LIN {X 0,Y 131.837,Z 270.712,A -85,B 0,C 180,E1 -26196.961,E2 -26196.961} C_VEL
LIN {X 0,Y 133.527,Z 251.929,A -85,B 0,C 180,E1 -26198.085,E2 -26198.085} C_VEL
LIN {X 0,Y 135.598,Z 225.127,A -85,B 0,C 180,E1 -26199.486,E2 -26199.486} C_VEL
LIN {X 0,Y 130.645,Z 212.931,A -85,B 0,C 180,E1 -26202.013,E2 -26202.013} C_VEL
LIN {X 0,Y 122.665,Z 198.092,A -85,B 0,C 180,E1 -26206.231,E2 -26206.231} C_VEL
LIN {X 0,Y 115.926,Z 187.635,A -85,B 0,C 180,E1 -26210.225,E2 -26210.225} C_VEL
LIN {X 0,Y 113.416,Z 183.95,A -85,B 0,C 180,E1 -26211.866,E2 -26211.866} C_VEL
LIN {X 0,Y 111.206,Z 180.453,A -85,B 0,C 180,E1 -26213.445,E2 -26213.445} C_VEL
LIN {X 0,Y 108.659,Z 177.597,A -85,B 0,C 180,E1 -26215.273,E2 -26215.273} C_VEL
LIN {X 0,Y 107.799,Z 175.056,A -85,B 0,C 180,E1 -26216.159,E2 -26216.159} C_VEL
LIN {X 0,Y 107.779,Z 175.058,A -85,B 0,C 180,E1 -26222.039,E2 -26222.039} C_VEL
LIN {X 0,Y 107.684,Z 175.066,A -85,B 0,C 180,E1 -26228.449,E2 -26228.449} C_VEL
LIN {X 0,Y 107.678,Z 175.072,A -85,B 0,C 180,E1 -26235.886,E2 -26235.886} C_VEL
LIN {X 0,Y 107.705,Z 175.047,A -85,B 0,C 180,E1 -26241.538,E2 -26241.538} C_VEL
LIN {X 0,Y 107.802,Z 175.038,A -85,B 0,C 180,E1 -26248.565,E2 -26248.565} C_VEL
LIN {X 0,Y 107.911,Z 175.043,A -85,B 0,C 180,E1 -26256.999,E2 -26256.999} C_VEL
LIN {X 0,Y 108.039,Z 175.012,A -85,B 0,C 180,E1 -26264.919,E2 -26264.919} C_VEL
LIN {X 0,Y 108.288,Z 174.994,A -85,B 0,C 180,E1 -26268.773,E2 -26268.773} C_VEL
LIN {X 0,Y 108.457,Z 174.961,A -85,B 0,C 180,E1 -26276.285,E2 -26276.285} C_VEL
LIN {X 0,Y 108.945,Z 174.908,A -85,B 0,C 180,E1 -26280.001,E2 -26280.001} C_VEL
LIN {X 0,Y 108.329,Z 174.987,A -85,B 0,C 180,E1 -26287.456,E2 -26287.456} C_VEL
LIN {X 0,Y 108.2,Z 174.989,A -85,B 0,C 180,E1 -26293.017,E2 -26293.017} C_VEL
LIN {X 0,Y 107.908,Z 175.033,A -85,B 0,C 180,E1 -26299.006,E2 -26299.006} C_VEL
LIN {X 0,Y 107.848,Z 175.044,A -85,B 0,C 180,E1 -26305.296,E2 -26305.296} C_VEL
LIN {X 0,Y 107.812,Z 175.158,A -85,B 0,C 180,E1 -26305.994,E2 -26305.994} C_VEL
LIN {X 0,Y 108.749,Z 177.876,A -85,B 0,C 180,E1 -26306.897,E2 -26306.897} C_VEL
LIN {X 0,Y 110.862,Z 180.069,A -85,B 0,C 180,E1 -26308.39,E2 -26308.39} C_VEL
LIN {X 0,Y 113.377,Z 183.974,A -85,B 0,C 180,E1 -26310.189,E2 -26310.189} C_VEL
LIN {X 0,Y 116.979,Z 189.548,A -85,B 0,C 180,E1 -26312.553,E2 -26312.553} C_VEL
LIN {X 0,Y 121.423,Z 196.893,A -85,B 0,C 180,E1 -26315.224,E2 -26315.224} C_VEL
LIN {X 0,Y 126.867,Z 209.823,A -85,B 0,C 180,E1 -26318.489,E2 -26318.489} C_VEL
LIN {X 0,Y 131.896,Z 223.796,A -85,B 0,C 180,E1 -26321.338,E2 -26321.338} C_VEL
LIN {X 0,Y 133.622,Z 229.369,A -85,B 0,C 180,E1 -26322.318,E2 -26322.318} C_VEL
LIN {X 0,Y 134.484,Z 244.81,A -85,B 0,C 180,E1 -26323.749,E2 -26323.749} C_VEL
LIN {X 0,Y 131.522,Z 280.67,A -85,B 0,C 180,E1 -26325.705,E2 -26325.705} C_VEL
LIN {X 0,Y 129.707,Z 293.105,A -85,B 0,C 180,E1 -26326.838,E2 -26326.838} C_VEL
LIN {X 0,Y 126.95,Z 306.45,A -85,B 0,C 180,E1 -26328.634,E2 -26328.634} C_VEL
LIN {X 0,Y 123.797,Z 318.083,A -85,B 0,C 180,E1 -26330.834,E2 -26330.834} C_VEL
LIN {X 0,Y 120.243,Z 329.412,A -85,B 0,C 180,E1 -26333.716,E2 -26333.716} C_VEL
LIN {X 0,Y 116.614,Z 339.667,A -85,B 0,C 180,E1 -26337.153,E2 -26337.153} C_VEL
LIN {X 0,Y 113.178,Z 348.906,A -85,B 0,C 180,E1 -26341.233,E2 -26341.233} C_VEL
LIN {X 0,Y 109.944,Z 357.92,A -85,B 0,C 180,E1 -26346.452,E2 -26346.452} C_VEL
LIN {X 0,Y 107.523,Z 365.11,A -85,B 0,C 180,E1 -26351.912,E2 -26351.912} C_VEL
LIN {X 0,Y 105.953,Z 371.622,A -85,B 0,C 180,E1 -26358.522,E2 -26358.522} C_VEL
LIN {X 0,Y 105.611,Z 375.867,A -85,B 0,C 180,E1 -26364.271,E2 -26364.271} C_VEL
LIN {X 0,Y 105.837,Z 378.956,A -85,B 0,C 180,E1 -26370,E2 -26370} C_VEL
LIN {X 0,Y 105.526,Z 380.371,A -85,B 0,C 180,E1 -26373.818,E2 -26373.818} C_VEL
LIN {X 0,Y 105.444,Z 381.376,A -85,B 0,C 180,E1 -26377.66,E2 -26377.66} C_VEL
LIN {X 0,Y 106.579,Z 382.189,A -85,B 0,C 180,E1 -26385.293,E2 -26385.293} C_VEL
LIN {X 0,Y 109.574,Z 381.541,A -85,B 0,C 180,E1 -26392.633,E2 -26392.633} C_VEL
LIN {X 0,Y 114.392,Z 379.409,A -85,B 0,C 180,E1 -26399.439,E2 -26399.439} C_VEL
LIN {X 0,Y 120.75,Z 375.708,A -85,B 0,C 180,E1 -26405.593,E2 -26405.593} C_VEL
LIN {X 0,Y 126.372,Z 371.837,A -85,B 0,C 180,E1 -26409.758,E2 -26409.758} C_VEL
LIN {X 0,Y 132.761,Z 366.913,A -85,B 0,C 180,E1 -26413.486,E2 -26413.486} C_VEL
LIN {X 0,Y 140.925,Z 359.728,A -85,B 0,C 180,E1 -26417.357,E2 -26417.357} C_VEL
LIN {X 0,Y 148.839,Z 351.65,A -85,B 0,C 180,E1 -26420.348,E2 -26420.348} C_VEL
LIN {X 0,Y 156.514,Z 342.43,A -85,B 0,C 180,E1 -26422.847,E2 -26422.847} C_VEL
LIN {X 0,Y 163.463,Z 332.667,A -85,B 0,C 180,E1 -26424.774,E2 -26424.774} C_VEL
LIN {X 0,Y 165.572,Z 329.353,A -85,B 0,C 180,E1 -26425.287,E2 -26425.287} C_VEL
LIN {X 0,Y 168.177,Z 324.681,A -85,B 0,C 180,E1 -26426.147,E2 -26426.147} C_VEL
LIN {X 0,Y 171.358,Z 317.027,A -85,B 0,C 180,E1 -26427.987,E2 -26427.987} C_VEL
LIN {X 0,Y 174.237,Z 309.028,A -85,B 0,C 180,E1 -26429.66,E2 -26429.66} C_VEL
LIN {X 0,Y 176.217,Z 303.822,A -85,B 0,C 180,E1 -26430.28,E2 -26430.28} C_VEL
LIN {X 0,Y 180.185,Z 292.508,A -85,B 0,C 180,E1 -26431,E2 -26431} C_VEL
LIN {X 0,Y 183.545,Z 279.289,A -85,B 0,C 180,E1 -26431.581,E2 -26431.581} C_VEL
LIN {X 0,Y 184.874,Z 271.488,A -85,B 0,C 180,E1 -26431.877,E2 -26431.877} C_VEL
LIN {X 0,Y 184.085,Z 267.5,A -85,B 0,C 180,E1 -26434.147,E2 -26434.147} C_VEL
LIN {X 0,Y 183.505,Z 264.746,A -85,B 0,C 180,E1 -26436.214,E2 -26436.214} C_VEL
LIN {X 0,Y 183.071,Z 262.291,A -85,B 0,C 180,E1 -26438.789,E2 -26438.789} C_VEL
LIN {X 0,Y 182.897,Z 261.223,A -85,B 0,C 180,E1 -26441.141,E2 -26441.141} C_VEL
LIN {X 0,Y 183.287,Z 261.303,A -85,B 0,C 180,E1 -26445.419,E2 -26445.419} C_VEL
LIN {X 0,Y 184.804,Z 265.34,A -85,B 0,C 180,E1 -26450.463,E2 -26450.463} C_VEL
LIN {X 0,Y 185.328,Z 267.395,A -85,B 0,C 180,E1 -26451.844,E2 -26451.844} C_VEL
LIN {X 0,Y 182.72,Z 280.977,A -85,B 0,C 180,E1 -26452.43,E2 -26452.43} C_VEL
LIN {X 0,Y 179.105,Z 293.413,A -85,B 0,C 180,E1 -26453.239,E2 -26453.239} C_VEL
LIN {X 0,Y 174.048,Z 306.258,A -85,B 0,C 180,E1 -26454.437,E2 -26454.437} C_VEL
LIN {X 0,Y 168.223,Z 317.797,A -85,B 0,C 180,E1 -26455.895,E2 -26455.895} C_VEL
LIN {X 0,Y 161.224,Z 328.841,A -85,B 0,C 180,E1 -26457.736,E2 -26457.736} C_VEL
LIN {X 0,Y 154.617,Z 337.56,A -85,B 0,C 180,E1 -26459.691,E2 -26459.691} C_VEL
LIN {X 0,Y 146.318,Z 346.778,A -85,B 0,C 180,E1 -26462.502,E2 -26462.502} C_VEL
LIN {X 0,Y 137.818,Z 354.628,A -85,B 0,C 180,E1 -26465.853,E2 -26465.853} C_VEL
LIN {X 0,Y 130.525,Z 360.305,A -85,B 0,C 180,E1 -26469.295,E2 -26469.295} C_VEL
LIN {X 0,Y 122.931,Z 365.24,A -85,B 0,C 180,E1 -26473.619,E2 -26473.619} C_VEL
LIN {X 0,Y 117.561,Z 368.123,A -85,B 0,C 180,E1 -26477.391,E2 -26477.391} C_VEL
LIN {X 0,Y 112.094,Z 370.491,A -85,B 0,C 180,E1 -26482.097,E2 -26482.097} C_VEL
LIN {X 0,Y 107.426,Z 371.92,A -85,B 0,C 180,E1 -26487.254,E2 -26487.254} C_VEL
LIN {X 0,Y 102.613,Z 372.423,A -85,B 0,C 180,E1 -26494.727,E2 -26494.727} C_VEL
LIN {X 0,Y 100.442,Z 371.896,A -85,B 0,C 180,E1 -26499.676,E2 -26499.676} C_VEL
LIN {X 0,Y 98.797,Z 370.594,A -85,B 0,C 180,E1 -26505.344,E2 -26505.344} C_VEL
LIN {X 0,Y 97.987,Z 368.076,A -85,B 0,C 180,E1 -26512.088,E2 -26512.088} C_VEL
LIN {X 0,Y 98.357,Z 364.286,A -85,B 0,C 180,E1 -26519.029,E2 -26519.029} C_VEL
LIN {X 0,Y 99.859,Z 358.869,A -85,B 0,C 180,E1 -26526.194,E2 -26526.194} C_VEL
LIN {X 0,Y 102.179,Z 351.971,A -85,B 0,C 180,E1 -26532.88,E2 -26532.88} C_VEL
LIN {X 0,Y 105.096,Z 344.444,A -85,B 0,C 180,E1 -26538.427,E2 -26538.427} C_VEL
LIN {X 0,Y 108.652,Z 335.44,A -85,B 0,C 180,E1 -26543.501,E2 -26543.501} C_VEL
LIN {X 0,Y 111.955,Z 326.806,A -85,B 0,C 180,E1 -26547.252,E2 -26547.252} C_VEL
LIN {X 0,Y 115.723,Z 316.032,A -85,B 0,C 180,E1 -26550.87,E2 -26550.87} C_VEL
LIN {X 0,Y 119.401,Z 303.884,A -85,B 0,C 180,E1 -26553.946,E2 -26553.946} C_VEL
LIN {X 0,Y 122.429,Z 291.632,A -85,B 0,C 180,E1 -26556.21,E2 -26556.21} C_VEL
LIN {X 0,Y 124.862,Z 278.393,A -85,B 0,C 180,E1 -26557.988,E2 -26557.988} C_VEL
LIN {X 0,Y 126.521,Z 265.545,A -85,B 0,C 180,E1 -26559.089,E2 -26559.089} C_VEL
LIN {X 0,Y 129.685,Z 227.021,A -85,B 0,C 180,E1 -26561.204,E2 -26561.204} C_VEL
LIN {X 0,Y 125.719,Z 217.007,A -85,B 0,C 180,E1 -26563.389,E2 -26563.389} C_VEL
LIN {X 0,Y 118.24,Z 202.715,A -85,B 0,C 180,E1 -26567.693,E2 -26567.693} C_VEL
LIN {X 0,Y 111.077,Z 191.405,A -85,B 0,C 180,E1 -26572.311,E2 -26572.311} C_VEL
LIN {X 0,Y 107.022,Z 185.413,A -85,B 0,C 180,E1 -26575.35,E2 -26575.35} C_VEL
LIN {X 0,Y 104.709,Z 182.294,A -85,B 0,C 180,E1 -26577.202,E2 -26577.202} C_VEL
LIN {X 0,Y 104.052,Z 181.117,A -85,B 0,C 180,E1 -26577.789,E2 -26577.789} C_VEL
LIN {X 0,Y 101.854,Z 179.084,A -85,B 0,C 180,E1 -26579.609,E2 -26579.609} C_VEL
LIN {X 0,Y 100.819,Z 176.566,A -85,B 0,C 180,E1 -26580.74,E2 -26580.74} C_VEL
LIN {X 0,Y 100.71,Z 175.936,A -85,B 0,C 180,E1 -26580.977,E2 -26580.977} C_VEL
LIN {X 0,Y 100.662,Z 175.944,A -85,B 0,C 180,E1 -26583.955,E2 -26583.955} C_VEL
LIN {X 0,Y 100.635,Z 175.933,A -85,B 0,C 180,E1 -26589.809,E2 -26589.809} C_VEL
LIN {X 0,Y 100.648,Z 175.947,A -85,B 0,C 180,E1 -26595.712,E2 -26595.712} C_VEL
LIN {X 0,Y 100.642,Z 175.924,A -85,B 0,C 180,E1 -26601.063,E2 -26601.063} C_VEL
LIN {X 0,Y 100.697,Z 175.936,A -85,B 0,C 180,E1 -26606.879,E2 -26606.879} C_VEL
LIN {X 0,Y 100.786,Z 175.928,A -85,B 0,C 180,E1 -26615.268,E2 -26615.268} C_VEL
LIN {X 0,Y 100.818,Z 175.909,A -85,B 0,C 180,E1 -26619.602,E2 -26619.602} C_VEL
LIN {X 0,Y 101.188,Z 175.879,A -85,B 0,C 180,E1 -26627.974,E2 -26627.974} C_VEL
LIN {X 0,Y 101.267,Z 175.844,A -85,B 0,C 180,E1 -26632.022,E2 -26632.022} C_VEL
LIN {X 0,Y 101.869,Z 175.788,A -85,B 0,C 180,E1 -26640.001,E2 -26640.001} C_VEL
LIN {X 0,Y 101.267,Z 175.868,A -85,B 0,C 180,E1 -26647.979,E2 -26647.979} C_VEL
LIN {X 0,Y 101.125,Z 175.87,A -85,B 0,C 180,E1 -26653.353,E2 -26653.353} C_VEL
LIN {X 0,Y 100.848,Z 176.055,A -85,B 0,C 180,E1 -26661.328,E2 -26661.328} C_VEL
LIN {X 0,Y 101.616,Z 178.356,A -85,B 0,C 180,E1 -26662.225,E2 -26662.225} C_VEL
LIN {X 0,Y 103.667,Z 180.769,A -85,B 0,C 180,E1 -26664.003,E2 -26664.003} C_VEL
LIN {X 0,Y 104.515,Z 181.953,A -85,B 0,C 180,E1 -26664.72,E2 -26664.72} C_VEL
LIN {X 0,Y 106.599,Z 185.091,A -85,B 0,C 180,E1 -26666.426,E2 -26666.426} C_VEL
LIN {X 0,Y 107.746,Z 186.474,A -85,B 0,C 180,E1 -26667.3,E2 -26667.3} C_VEL
LIN {X 0,Y 112.889,Z 194.47,A -85,B 0,C 180,E1 -26671.036,E2 -26671.036} C_VEL
LIN {X 0,Y 116.945,Z 201.381,A -85,B 0,C 180,E1 -26673.685,E2 -26673.685} C_VEL
LIN {X 0,Y 122.57,Z 215.234,A -85,B 0,C 180,E1 -26677.347,E2 -26677.347} C_VEL
LIN {X 0,Y 127.889,Z 231.188,A -85,B 0,C 180,E1 -26680.607,E2 -26680.607} C_VEL
LIN {X 0,Y 128.625,Z 245.668,A -85,B 0,C 180,E1 -26682.015,E2 -26682.015} C_VEL
LIN {X 0,Y 125.645,Z 280.029,A -85,B 0,C 180,E1 -26683.932,E2 -26683.932} C_VEL
LIN {X 0,Y 123.808,Z 292.415,A -85,B 0,C 180,E1 -26685.089,E2 -26685.089} C_VEL
LIN {X 0,Y 121.183,Z 304.754,A -85,B 0,C 180,E1 -26686.76,E2 -26686.76} C_VEL
LIN {X 0,Y 117.888,Z 316.726,A -85,B 0,C 180,E1 -26689.022,E2 -26689.022} C_VEL
LIN {X 0,Y 114.118,Z 328.195,A -85,B 0,C 180,E1 -26691.986,E2 -26691.986} C_VEL
LIN {X 0,Y 110.296,Z 338.594,A -85,B 0,C 180,E1 -26695.564,E2 -26695.564} C_VEL
LIN {X 0,Y 107.001,Z 347.129,A -85,B 0,C 180,E1 -26699.401,E2 -26699.401} C_VEL
LIN {X 0,Y 103.905,Z 354.985,A -85,B 0,C 180,E1 -26703.918,E2 -26703.918} C_VEL
LIN {X 0,Y 101.156,Z 362.651,A -85,B 0,C 180,E1 -26709.673,E2 -26709.673} C_VEL
LIN {X 0,Y 99.349,Z 368.774,A -85,B 0,C 180,E1 -26715.665,E2 -26715.665} C_VEL
LIN {X 0,Y 98.608,Z 373.592,A -85,B 0,C 180,E1 -26721.805,E2 -26721.805} C_VEL
LIN {X 0,Y 98.604,Z 376.347,A -85,B 0,C 180,E1 -26726.256,E2 -26726.256} C_VEL
LIN {X 0,Y 98.775,Z 378.176,A -85,B 0,C 180,E1 -26730,E2 -26730} C_VEL
LIN {X 0,Y 98.468,Z 379.662,A -85,B 0,C 180,E1 -26734.093,E2 -26734.093} C_VEL
LIN {X 0,Y 98.827,Z 381.446,A -85,B 0,C 180,E1 -26742.318,E2 -26742.318} C_VEL
LIN {X 0,Y 101.069,Z 381.683,A -85,B 0,C 180,E1 -26750.345,E2 -26750.345} C_VEL
LIN {X 0,Y 105.411,Z 380.472,A -85,B 0,C 180,E1 -26757.82,E2 -26757.82} C_VEL
LIN {X 0,Y 111.463,Z 377.78,A -85,B 0,C 180,E1 -26764.574,E2 -26764.574} C_VEL
LIN {X 0,Y 118.938,Z 373.459,A -85,B 0,C 180,E1 -26770.54,E2 -26770.54} C_VEL
LIN {X 0,Y 125.397,Z 369.107,A -85,B 0,C 180,E1 -26774.473,E2 -26774.473} C_VEL
LIN {X 0,Y 133.757,Z 362.639,A -85,B 0,C 180,E1 -26778.481,E2 -26778.481} C_VEL
LIN {X 0,Y 140.203,Z 356.907,A -85,B 0,C 180,E1 -26780.983,E2 -26780.983} C_VEL
LIN {X 0,Y 148.219,Z 348.662,A -85,B 0,C 180,E1 -26783.714,E2 -26783.714} C_VEL
LIN {X 0,Y 155.241,Z 340.323,A -85,B 0,C 180,E1 -26785.71,E2 -26785.71} C_VEL
LIN {X 0,Y 162.487,Z 330.174,A -85,B 0,C 180,E1 -26787.503,E2 -26787.503} C_VEL
LIN {X 0,Y 169.161,Z 318.917,A -85,B 0,C 180,E1 -26788.968,E2 -26788.968} C_VEL
LIN {X 0,Y 174.516,Z 307.935,A -85,B 0,C 180,E1 -26789.977,E2 -26789.977} C_VEL
LIN {X 0,Y 176.217,Z 303.822,A -85,B 0,C 180,E1 -26790.28,E2 -26790.28} C_VEL
LIN {X 0,Y 177.445,Z 300.288,A -85,B 0,C 180,E1 -26790.733,E2 -26790.733} C_VEL
LIN {X 0,Y 178.72,Z 294.85,A -85,B 0,C 180,E1 -26791.96,E2 -26791.96} C_VEL
LIN {X 0,Y 179.777,Z 289.299,A -85,B 0,C 180,E1 -26793.142,E2 -26793.142} C_VEL
LIN {X 0,Y 180.602,Z 285.59,A -85,B 0,C 180,E1 -26793.524,E2 -26793.524} C_VEL
LIN {X 0,Y 182.811,Z 275.727,A -85,B 0,C 180,E1 -26793.867,E2 -26793.867} C_VEL
LIN {X 0,Y 182.294,Z 271.985,A -85,B 0,C 180,E1 -26796.36,E2 -26796.36} C_VEL
LIN {X 0,Y 181.952,Z 269.208,A -85,B 0,C 180,E1 -26799.156,E2 -26799.156} C_VEL
LIN {X 0,Y 181.841,Z 268.21,A -85,B 0,C 180,E1 -26801.337,E2 -26801.337} C_VEL
LIN {X 0,Y 182.176,Z 268.432,A -85,B 0,C 180,E1 -26805.328,E2 -26805.328} C_VEL
LIN {X 0,Y 183.288,Z 271.943,A -85,B 0,C 180,E1 -26809.815,E2 -26809.815} C_VEL
LIN {X 0,Y 180.017,Z 285.949,A -85,B 0,C 180,E1 -26810.494,E2 -26810.494} C_VEL
LIN {X 0,Y 175.935,Z 298.146,A -85,B 0,C 180,E1 -26811.366,E2 -26811.366} C_VEL
LIN {X 0,Y 171.04,Z 309.246,A -85,B 0,C 180,E1 -26812.43,E2 -26812.43} C_VEL
LIN {X 0,Y 164.303,Z 321.376,A -85,B 0,C 180,E1 -26813.99,E2 -26813.99} C_VEL
LIN {X 0,Y 157.491,Z 331.354,A -85,B 0,C 180,E1 -26815.691,E2 -26815.691} C_VEL
LIN {X 0,Y 150.36,Z 340.057,A -85,B 0,C 180,E1 -26817.691,E2 -26817.691} C_VEL
LIN {X 0,Y 142.414,Z 348.233,A -85,B 0,C 180,E1 -26820.233,E2 -26820.233} C_VEL
LIN {X 0,Y 133.771,Z 355.686,A -85,B 0,C 180,E1 -26823.437,E2 -26823.437} C_VEL
LIN {X 0,Y 127.087,Z 360.535,A -85,B 0,C 180,E1 -26826.349,E2 -26826.349} C_VEL
LIN {X 0,Y 119.824,Z 365.053,A -85,B 0,C 180,E1 -26830.134,E2 -26830.134} C_VEL
LIN {X 0,Y 113.211,Z 368.442,A -85,B 0,C 180,E1 -26834.377,E2 -26834.377} C_VEL
LIN {X 0,Y 107.19,Z 370.854,A -85,B 0,C 180,E1 -26839.136,E2 -26839.136} C_VEL
LIN {X 0,Y 101.17,Z 372.491,A -85,B 0,C 180,E1 -26845.436,E2 -26845.436} C_VEL
LIN {X 0,Y 97.679,Z 372.854,A -85,B 0,C 180,E1 -26850.301,E2 -26850.301} C_VEL
LIN {X 0,Y 94.409,Z 372.476,A -85,B 0,C 180,E1 -26856.55,E2 -26856.55} C_VEL
LIN {X 0,Y 92.072,Z 371.103,A -85,B 0,C 180,E1 -26863.39,E2 -26863.39} C_VEL
LIN {X 0,Y 90.92,Z 368.136,A -85,B 0,C 180,E1 -26871.802,E2 -26871.802} C_VEL
LIN {X 0,Y 91.435,Z 363.55,A -85,B 0,C 180,E1 -26880.359,E2 -26880.359} C_VEL
LIN {X 0,Y 93.118,Z 357.907,A -85,B 0,C 180,E1 -26887.829,E2 -26887.829} C_VEL
LIN {X 0,Y 95.204,Z 352.116,A -85,B 0,C 180,E1 -26893.669,E2 -26893.669} C_VEL
LIN {X 0,Y 98.322,Z 344.497,A -85,B 0,C 180,E1 -26899.605,E2 -26899.605} C_VEL
LIN {X 0,Y 102.172,Z 335.189,A -85,B 0,C 180,E1 -26905.068,E2 -26905.068} C_VEL
LIN {X 0,Y 106.043,Z 325.472,A -85,B 0,C 180,E1 -26909.369,E2 -26909.369} C_VEL
LIN {X 0,Y 110.176,Z 313.999,A -85,B 0,C 180,E1 -26913.2,E2 -26913.2} C_VEL
LIN {X 0,Y 113.931,Z 301.728,A -85,B 0,C 180,E1 -26916.203,E2 -26916.203} C_VEL
LIN {X 0,Y 116.91,Z 289.5,A -85,B 0,C 180,E1 -26918.426,E2 -26918.426} C_VEL
LIN {X 0,Y 119.334,Z 276.391,A -85,B 0,C 180,E1 -26920.069,E2 -26920.069} C_VEL
LIN {X 0,Y 120.936,Z 263.248,A -85,B 0,C 180,E1 -26921.138,E2 -26921.138} C_VEL
LIN {X 0,Y 123.884,Z 229.049,A -85,B 0,C 180,E1 -26923.032,E2 -26923.032} C_VEL
LIN {X 0,Y 120.908,Z 221.221,A -85,B 0,C 180,E1 -26924.852,E2 -26924.852} C_VEL
LIN {X 0,Y 113.931,Z 207.494,A -85,B 0,C 180,E1 -26929.179,E2 -26929.179} C_VEL
LIN {X 0,Y 107.162,Z 196.422,A -85,B 0,C 180,E1 -26933.971,E2 -26933.971} C_VEL
LIN {X 0,Y 103.405,Z 190.856,A -85,B 0,C 180,E1 -26936.984,E2 -26936.984} C_VEL
LIN {X 0,Y 100.54,Z 186.845,A -85,B 0,C 180,E1 -26939.521,E2 -26939.521} C_VEL
LIN {X 0,Y 98.208,Z 183.934,A -85,B 0,C 180,E1 -26941.766,E2 -26941.766} C_VEL
LIN {X 0,Y 97.345,Z 182.199,A -85,B 0,C 180,E1 -26942.753,E2 -26942.753} C_VEL
LIN {X 0,Y 94.812,Z 180.065,A -85,B 0,C 180,E1 -26945.376,E2 -26945.376} C_VEL
LIN {X 0,Y 93.678,Z 177.738,A -85,B 0,C 180,E1 -26946.883,E2 -26946.883} C_VEL
LIN {X 0,Y 93.528,Z 176.835,A -85,B 0,C 180,E1 -26947.215,E2 -26947.215} C_VEL
LIN {X 0,Y 93.53,Z 176.817,A -85,B 0,C 180,E1 -26952.553,E2 -26952.553} C_VEL
LIN {X 0,Y 93.542,Z 176.812,A -85,B 0,C 180,E1 -26958.705,E2 -26958.705} C_VEL
LIN {X 0,Y 93.596,Z 176.825,A -85,B 0,C 180,E1 -26965.687,E2 -26965.687} C_VEL
LIN {X 0,Y 93.668,Z 176.808,A -85,B 0,C 180,E1 -26974.206,E2 -26974.206} C_VEL
LIN {X 0,Y 93.695,Z 176.809,A -85,B 0,C 180,E1 -26977.974,E2 -26977.974} C_VEL
LIN {X 0,Y 94.092,Z 176.762,A -85,B 0,C 180,E1 -26987.052,E2 -26987.052} C_VEL
LIN {X 0,Y 94.2,Z 176.727,A -85,B 0,C 180,E1 -26991.42,E2 -26991.42} C_VEL
LIN {X 0,Y 94.795,Z 176.669,A -85,B 0,C 180,E1 -27000.001,E2 -27000.001} C_VEL
LIN {X 0,Y 94.2,Z 176.749,A -85,B 0,C 180,E1 -27008.582,E2 -27008.582} C_VEL
LIN {X 0,Y 94.043,Z 176.753,A -85,B 0,C 180,E1 -27013.71,E2 -27013.71} C_VEL
LIN {X 0,Y 93.921,Z 176.779,A -85,B 0,C 180,E1 -27015.239,E2 -27015.239} C_VEL
LIN {X 0,Y 94.772,Z 179.516,A -85,B 0,C 180,E1 -27016.58,E2 -27016.58} C_VEL
LIN {X 0,Y 96.82,Z 181.794,A -85,B 0,C 180,E1 -27018.846,E2 -27018.846} C_VEL
LIN {X 0,Y 97.701,Z 182.55,A -85,B 0,C 180,E1 -27019.72,E2 -27019.72} C_VEL
LIN {X 0,Y 99.712,Z 185.824,A -85,B 0,C 180,E1 -27021.812,E2 -27021.812} C_VEL
LIN {X 0,Y 101.077,Z 187.521,A -85,B 0,C 180,E1 -27023.061,E2 -27023.061} C_VEL
LIN {X 0,Y 103.594,Z 191.152,A -85,B 0,C 180,E1 -27025.259,E2 -27025.259} C_VEL
LIN {X 0,Y 108.523,Z 198.823,A -85,B 0,C 180,E1 -27029.176,E2 -27029.176} C_VEL
LIN {X 0,Y 112.552,Z 205.973,A -85,B 0,C 180,E1 -27032.064,E2 -27032.064} C_VEL
LIN {X 0,Y 117.632,Z 218.956,A -85,B 0,C 180,E1 -27035.67,E2 -27035.67} C_VEL
LIN {X 0,Y 122.271,Z 233.328,A -85,B 0,C 180,E1 -27038.821,E2 -27038.821} C_VEL
LIN {X 0,Y 122.836,Z 246.355,A -85,B 0,C 180,E1 -27040.147,E2 -27040.147} C_VEL
LIN {X 0,Y 119.807,Z 279.685,A -85,B 0,C 180,E1 -27042.062,E2 -27042.062} C_VEL
LIN {X 0,Y 117.896,Z 292.046,A -85,B 0,C 180,E1 -27043.249,E2 -27043.249} C_VEL
LIN {X 0,Y 115.019,Z 304.913,A -85,B 0,C 180,E1 -27045.049,E2 -27045.049} C_VEL
LIN {X 0,Y 111.577,Z 316.722,A -85,B 0,C 180,E1 -27047.381,E2 -27047.381} C_VEL
LIN {X 0,Y 107.656,Z 328.13,A -85,B 0,C 180,E1 -27050.469,E2 -27050.469} C_VEL
LIN {X 0,Y 103.913,Z 337.83,A -85,B 0,C 180,E1 -27053.956,E2 -27053.956} C_VEL
LIN {X 0,Y 100.188,Z 346.954,A -85,B 0,C 180,E1 -27058.257,E2 -27058.257} C_VEL
LIN {X 0,Y 96.965,Z 354.77,A -85,B 0,C 180,E1 -27063.064,E2 -27063.064} C_VEL
LIN {X 0,Y 94.102,Z 362.404,A -85,B 0,C 180,E1 -27069.222,E2 -27069.222} C_VEL
LIN {X 0,Y 92.03,Z 369.403,A -85,B 0,C 180,E1 -27076.756,E2 -27076.756} C_VEL
LIN {X 0,Y 91.509,Z 373.989,A -85,B 0,C 180,E1 -27083.385,E2 -27083.385} C_VEL
LIN {X 0,Y 91.716,Z 377.385,A -85,B 0,C 180,E1 -27090,E2 -27090} C_VEL
LIN {X 0,Y 91.404,Z 378.952,A -85,B 0,C 180,E1 -27094.41,E2 -27094.41} C_VEL
LIN {X 0,Y 91.893,Z 380.865,A -85,B 0,C 180,E1 -27103.264,E2 -27103.264} C_VEL
LIN {X 0,Y 94.412,Z 381.317,A -85,B 0,C 180,E1 -27111.851,E2 -27111.851} C_VEL
LIN {X 0,Y 99.156,Z 380.266,A -85,B 0,C 180,E1 -27119.745,E2 -27119.745} C_VEL
LIN {X 0,Y 105.67,Z 377.765,A -85,B 0,C 180,E1 -27126.768,E2 -27126.768} C_VEL
LIN {X 0,Y 111.513,Z 374.861,A -85,B 0,C 180,E1 -27131.433,E2 -27131.433} C_VEL
LIN {X 0,Y 118.099,Z 371.02,A -85,B 0,C 180,E1 -27135.57,E2 -27135.57} C_VEL
LIN {X 0,Y 125.363,Z 366.137,A -85,B 0,C 180,E1 -27139.184,E2 -27139.184} C_VEL
LIN {X 0,Y 134.494,Z 358.98,A -85,B 0,C 180,E1 -27142.833,E2 -27142.833} C_VEL
LIN {X 0,Y 142.768,Z 351.325,A -85,B 0,C 180,E1 -27145.542,E2 -27145.542} C_VEL
LIN {X 0,Y 151.418,Z 341.848,A -85,B 0,C 180,E1 -27147.893,E2 -27147.893} C_VEL
LIN {X 0,Y 158.84,Z 332.187,A -85,B 0,C 180,E1 -27149.631,E2 -27149.631} C_VEL
LIN {X 0,Y 165.668,Z 321.535,A -85,B 0,C 180,E1 -27151.039,E2 -27151.039} C_VEL
LIN {X 0,Y 171.924,Z 309.546,A -85,B 0,C 180,E1 -27152.127,E2 -27152.127} C_VEL
LIN {X 0,Y 176.95,Z 297.352,A -85,B 0,C 180,E1 -27152.95,E2 -27152.95} C_VEL
LIN {X 0,Y 180.602,Z 285.59,A -85,B 0,C 180,E1 -27153.524,E2 -27153.524} C_VEL
LIN {X 0,Y 181.053,Z 283.275,A -85,B 0,C 180,E1 -27153.816,E2 -27153.816} C_VEL
LIN {X 0,Y 181.299,Z 280.516,A -85,B 0,C 180,E1 -27154.69,E2 -27154.69} C_VEL
LIN {X 0,Y 181.208,Z 278.649,A -85,B 0,C 180,E1 -27155.82,E2 -27155.82} C_VEL
LIN {X 0,Y 180.861,Z 277.048,A -85,B 0,C 180,E1 -27157.668,E2 -27157.668} C_VEL
LIN {X 0,Y 180.594,Z 276.061,A -85,B 0,C 180,E1 -27159.571,E2 -27159.571} C_VEL
LIN {X 0,Y 180.543,Z 275.118,A -85,B 0,C 180,E1 -27161.855,E2 -27161.855} C_VEL
LIN {X 0,Y 180.787,Z 275.323,A -85,B 0,C 180,E1 -27164.934,E2 -27164.934} C_VEL
LIN {X 0,Y 181.138,Z 277.468,A -85,B 0,C 180,E1 -27167.834,E2 -27167.834} C_VEL
LIN {X 0,Y 177.546,Z 290.419,A -85,B 0,C 180,E1 -27168.487,E2 -27168.487} C_VEL
LIN {X 0,Y 172.711,Z 303.115,A -85,B 0,C 180,E1 -27169.453,E2 -27169.453} C_VEL
LIN {X 0,Y 167.048,Z 314.468,A -85,B 0,C 180,E1 -27170.597,E2 -27170.597} C_VEL
LIN {X 0,Y 159.834,Z 325.993,A -85,B 0,C 180,E1 -27172.167,E2 -27172.167} C_VEL
LIN {X 0,Y 152.293,Z 335.815,A -85,B 0,C 180,E1 -27173.942,E2 -27173.942} C_VEL
LIN {X 0,Y 144.403,Z 344.369,A -85,B 0,C 180,E1 -27176.1,E2 -27176.1} C_VEL
LIN {X 0,Y 135.31,Z 352.612,A -85,B 0,C 180,E1 -27178.949,E2 -27178.949} C_VEL
LIN {X 0,Y 126.595,Z 359.158,A -85,B 0,C 180,E1 -27182.185,E2 -27182.185} C_VEL
LIN {X 0,Y 117.874,Z 364.507,A -85,B 0,C 180,E1 -27186.148,E2 -27186.148} C_VEL
LIN {X 0,Y 109.149,Z 368.777,A -85,B 0,C 180,E1 -27191.137,E2 -27191.137} C_VEL
LIN {X 0,Y 102.399,Z 371.291,A -85,B 0,C 180,E1 -27196.083,E2 -27196.083} C_VEL
LIN {X 0,Y 96.89,Z 372.706,A -85,B 0,C 180,E1 -27201.264,E2 -27201.264} C_VEL
LIN {X 0,Y 92.065,Z 373.278,A -85,B 0,C 180,E1 -27207.259,E2 -27207.259} C_VEL
LIN {X 0,Y 87.178,Z 372.61,A -85,B 0,C 180,E1 -27216.278,E2 -27216.278} C_VEL
LIN {X 0,Y 85.238,Z 371.357,A -85,B 0,C 180,E1 -27222.093,E2 -27222.093} C_VEL
LIN {X 0,Y 83.855,Z 368.194,A -85,B 0,C 180,E1 -27231.453,E2 -27231.453} C_VEL
LIN {X 0,Y 84.247,Z 363.882,A -85,B 0,C 180,E1 -27239.965,E2 -27239.965} C_VEL
LIN {X 0,Y 86.089,Z 357.908,A -85,B 0,C 180,E1 -27248.447,E2 -27248.447} C_VEL
LIN {X 0,Y 88.461,Z 351.753,A -85,B 0,C 180,E1 -27255.003,E2 -27255.003} C_VEL
LIN {X 0,Y 91.732,Z 344.168,A -85,B 0,C 180,E1 -27261.186,E2 -27261.186} C_VEL
LIN {X 0,Y 95.786,Z 334.877,A -85,B 0,C 180,E1 -27266.847,E2 -27266.847} C_VEL
LIN {X 0,Y 99.568,Z 325.874,A -85,B 0,C 180,E1 -27271.011,E2 -27271.011} C_VEL
LIN {X 0,Y 103.634,Z 315.294,A -85,B 0,C 180,E1 -27274.743,E2 -27274.743} C_VEL
LIN {X 0,Y 107.094,Z 304.825,A -85,B 0,C 180,E1 -27277.542,E2 -27277.542} C_VEL
LIN {X 0,Y 110.619,Z 291.903,A -85,B 0,C 180,E1 -27280.062,E2 -27280.062} C_VEL
LIN {X 0,Y 113.257,Z 278.709,A -85,B 0,C 180,E1 -27281.912,E2 -27281.912} C_VEL
LIN {X 0,Y 115.149,Z 264.704,A -85,B 0,C 180,E1 -27283.129,E2 -27283.129} C_VEL
LIN {X 0,Y 118.288,Z 231.05,A -85,B 0,C 180,E1 -27285.012,E2 -27285.012} C_VEL
LIN {X 0,Y 115.756,Z 224.491,A -85,B 0,C 180,E1 -27286.688,E2 -27286.688} C_VEL
LIN {X 0,Y 109.296,Z 211.508,A -85,B 0,C 180,E1 -27291.076,E2 -27291.076} C_VEL
LIN {X 0,Y 102.552,Z 200.204,A -85,B 0,C 180,E1 -27296.364,E2 -27296.364} C_VEL
LIN {X 0,Y 99.616,Z 195.931,A -85,B 0,C 180,E1 -27298.958,E2 -27298.958} C_VEL
LIN {X 0,Y 97.292,Z 192.527,A -85,B 0,C 180,E1 -27301.247,E2 -27301.247} C_VEL
LIN {X 0,Y 94.853,Z 189.078,A -85,B 0,C 180,E1 -27303.88,E2 -27303.88} C_VEL
LIN {X 0,Y 94.085,Z 188.077,A -85,B 0,C 180,E1 -27304.748,E2 -27304.748} C_VEL
LIN {X 0,Y 91.686,Z 185.396,A -85,B 0,C 180,E1 -27307.588,E2 -27307.588} C_VEL
LIN {X 0,Y 90.627,Z 183.265,A -85,B 0,C 180,E1 -27309.152,E2 -27309.152} C_VEL
LIN {X 0,Y 87.911,Z 181.19,A -85,B 0,C 180,E1 -27312.993,E2 -27312.993} C_VEL
LIN {X 0,Y 86.65,Z 178.859,A -85,B 0,C 180,E1 -27315.349,E2 -27315.349} C_VEL
LIN {X 0,Y 86.427,Z 177.718,A -85,B 0,C 180,E1 -27316.021,E2 -27316.021} C_VEL
LIN {X 0,Y 86.463,Z 177.689,A -85,B 0,C 180,E1 -27319.44,E2 -27319.44} C_VEL
LIN {X 0,Y 86.54,Z 177.703,A -85,B 0,C 180,E1 -27325.357,E2 -27325.357} C_VEL
LIN {X 0,Y 86.583,Z 177.679,A -85,B 0,C 180,E1 -27333.237,E2 -27333.237} C_VEL
LIN {X 0,Y 86.648,Z 177.661,A -85,B 0,C 180,E1 -27341.069,E2 -27341.069} C_VEL
LIN {X 0,Y 86.97,Z 177.642,A -85,B 0,C 180,E1 -27345.971,E2 -27345.971} C_VEL
LIN {X 0,Y 87.108,Z 177.615,A -85,B 0,C 180,E1 -27350.715,E2 -27350.715} C_VEL
LIN {X 0,Y 87.722,Z 177.549,A -85,B 0,C 180,E1 -27360.001,E2 -27360.001} C_VEL
LIN {X 0,Y 87.172,Z 177.735,A -85,B 0,C 180,E1 -27367.238,E2 -27367.238} C_VEL
LIN {X 0,Y 87.942,Z 180.163,A -85,B 0,C 180,E1 -27368.908,E2 -27368.908} C_VEL
LIN {X 0,Y 89.658,Z 182.31,A -85,B 0,C 180,E1 -27371.589,E2 -27371.589} C_VEL
LIN {X 0,Y 91.165,Z 183.525,A -85,B 0,C 180,E1 -27373.567,E2 -27373.567} C_VEL
LIN {X 0,Y 92.884,Z 186.668,A -85,B 0,C 180,E1 -27375.92,E2 -27375.92} C_VEL
LIN {X 0,Y 94.959,Z 188.943,A -85,B 0,C 180,E1 -27378.298,E2 -27378.298} C_VEL
LIN {X 0,Y 98.258,Z 193.946,A -85,B 0,C 180,E1 -27381.828,E2 -27381.828} C_VEL
LIN {X 0,Y 101.569,Z 198.922,A -85,B 0,C 180,E1 -27384.892,E2 -27384.892} C_VEL
LIN {X 0,Y 105.148,Z 204.819,A -85,B 0,C 180,E1 -27387.897,E2 -27387.897} C_VEL
LIN {X 0,Y 108.223,Z 210.581,A -85,B 0,C 180,E1 -27390.324,E2 -27390.324} C_VEL
LIN {X 0,Y 112.7,Z 222.442,A -85,B 0,C 180,E1 -27393.811,E2 -27393.811} C_VEL
LIN {X 0,Y 116.887,Z 235.997,A -85,B 0,C 180,E1 -27396.961,E2 -27396.961} C_VEL
LIN {X 0,Y 117.203,Z 246.818,A -85,B 0,C 180,E1 -27398.092,E2 -27398.092} C_VEL
LIN {X 0,Y 114.088,Z 279.514,A -85,B 0,C 180,E1 -27400.022,E2 -27400.022} C_VEL
LIN {X 0,Y 112.101,Z 291.644,A -85,B 0,C 180,E1 -27401.208,E2 -27401.208} C_VEL
LIN {X 0,Y 108.957,Z 305.048,A -85,B 0,C 180,E1 -27403.14,E2 -27403.14} C_VEL
LIN {X 0,Y 105.39,Z 316.732,A -85,B 0,C 180,E1 -27405.557,E2 -27405.557} C_VEL
LIN {X 0,Y 101.281,Z 328.065,A -85,B 0,C 180,E1 -27408.76,E2 -27408.76} C_VEL
LIN {X 0,Y 97.44,Z 337.532,A -85,B 0,C 180,E1 -27412.338,E2 -27412.338} C_VEL
LIN {X 0,Y 93.425,Z 346.775,A -85,B 0,C 180,E1 -27416.949,E2 -27416.949} C_VEL
LIN {X 0,Y 89.516,Z 355.935,A -85,B 0,C 180,E1 -27423.164,E2 -27423.164} C_VEL
LIN {X 0,Y 86.63,Z 363.27,A -85,B 0,C 180,E1 -27429.831,E2 -27429.831} C_VEL
LIN {X 0,Y 85.119,Z 368.199,A -85,B 0,C 180,E1 -27435.659,E2 -27435.659} C_VEL
LIN {X 0,Y 84.462,Z 372.957,A -85,B 0,C 180,E1 -27442.83,E2 -27442.83} C_VEL
LIN {X 0,Y 84.657,Z 376.507,A -85,B 0,C 180,E1 -27450,E2 -27450} C_VEL
LIN {X 0,Y 84.341,Z 378.191,A -85,B 0,C 180,E1 -27454.78,E2 -27454.78} C_VEL
LIN {X 0,Y 84.996,Z 380.281,A -85,B 0,C 180,E1 -27464.362,E2 -27464.362} C_VEL
LIN {X 0,Y 87.835,Z 380.888,A -85,B 0,C 180,E1 -27473.582,E2 -27473.582} C_VEL
LIN {X 0,Y 93.031,Z 380.072,A -85,B 0,C 180,E1 -27481.925,E2 -27481.925} C_VEL
LIN {X 0,Y 100.041,Z 377.743,A -85,B 0,C 180,E1 -27489.217,E2 -27489.217} C_VEL
LIN {X 0,Y 108.525,Z 373.909,A -85,B 0,C 180,E1 -27495.426,E2 -27495.426} C_VEL
LIN {X 0,Y 115.725,Z 369.92,A -85,B 0,C 180,E1 -27499.386,E2 -27499.386} C_VEL
LIN {X 0,Y 123.558,Z 364.893,A -85,B 0,C 180,E1 -27502.779,E2 -27502.779} C_VEL
LIN {X 0,Y 130.358,Z 359.803,A -85,B 0,C 180,E1 -27505.302,E2 -27505.302} C_VEL
LIN {X 0,Y 138.921,Z 352.426,A -85,B 0,C 180,E1 -27507.927,E2 -27507.927} C_VEL
LIN {X 0,Y 147.825,Z 343.362,A -85,B 0,C 180,E1 -27510.186,E2 -27510.186} C_VEL
LIN {X 0,Y 156.2,Z 333.097,A -85,B 0,C 180,E1 -27512.005,E2 -27512.005} C_VEL
LIN {X 0,Y 163.209,Z 322.798,A -85,B 0,C 180,E1 -27513.318,E2 -27513.318} C_VEL
LIN {X 0,Y 169.599,Z 311.402,A -85,B 0,C 180,E1 -27514.328,E2 -27514.328} C_VEL
LIN {X 0,Y 175.154,Z 298.653,A -85,B 0,C 180,E1 -27515.158,E2 -27515.158} C_VEL
LIN {X 0,Y 179.468,Z 285.427,A -85,B 0,C 180,E1 -27515.764,E2 -27515.764} C_VEL
LIN {X 0,Y 180.802,Z 280.005,A -85,B 0,C 180,E1 -27515.984,E2 -27515.984} C_VEL
LIN {X 0,Y 180.604,Z 277.082,A -85,B 0,C 180,E1 -27518.449,E2 -27518.449} C_VEL
LIN {X 0,Y 180.594,Z 276.061,A -85,B 0,C 180,E1 -27519.571,E2 -27519.571} C_VEL
LIN {X 0,Y 180.357,Z 276.653,A -85,B 0,C 180,E1 -27520.324,E2 -27520.324} C_VEL
LIN {X 0,Y 179.035,Z 281.576,A -85,B 0,C 180,E1 -27522.14,E2 -27522.14} C_VEL
LIN {X 0,Y 178.916,Z 282.049,A -85,B 0,C 180,E1 -27522.706,E2 -27522.706} C_VEL
LIN {X 0,Y 179.061,Z 282.183,A -85,B 0,C 180,E1 -27524.602,E2 -27524.602} C_VEL
LIN {X 0,Y 179.059,Z 283.056,A -85,B 0,C 180,E1 -27525.792,E2 -27525.792} C_VEL
LIN {X 0,Y 175.126,Z 295.183,A -85,B 0,C 180,E1 -27526.491,E2 -27526.491} C_VEL
LIN {X 0,Y 169.728,Z 307.588,A -85,B 0,C 180,E1 -27527.454,E2 -27527.454} C_VEL
LIN {X 0,Y 164.038,Z 317.96,A -85,B 0,C 180,E1 -27528.532,E2 -27528.532} C_VEL
LIN {X 0,Y 157.034,Z 328.353,A -85,B 0,C 180,E1 -27529.928,E2 -27529.928} C_VEL
LIN {X 0,Y 149.177,Z 337.898,A -85,B 0,C 180,E1 -27531.627,E2 -27531.627} C_VEL
LIN {X 0,Y 139.907,Z 347.234,A -85,B 0,C 180,E1 -27534.002,E2 -27534.002} C_VEL
LIN {X 0,Y 131.686,Z 354.069,A -85,B 0,C 180,E1 -27536.412,E2 -27536.412} C_VEL
LIN {X 0,Y 121.434,Z 361.077,A -85,B 0,C 180,E1 -27539.999,E2 -27539.999} C_VEL
LIN {X 0,Y 112.694,Z 365.932,A -85,B 0,C 180,E1 -27543.797,E2 -27543.797} C_VEL
LIN {X 0,Y 105.5,Z 369.142,A -85,B 0,C 180,E1 -27547.656,E2 -27547.656} C_VEL
LIN {X 0,Y 98.409,Z 371.598,A -85,B 0,C 180,E1 -27552.37,E2 -27552.37} C_VEL
LIN {X 0,Y 92.116,Z 373.1,A -85,B 0,C 180,E1 -27557.768,E2 -27557.768} C_VEL
LIN {X 0,Y 85.59,Z 373.712,A -85,B 0,C 180,E1 -27565.415,E2 -27565.415} C_VEL
LIN {X 0,Y 82.116,Z 373.343,A -85,B 0,C 180,E1 -27571.146,E2 -27571.146} C_VEL
LIN {X 0,Y 79.041,Z 372.1,A -85,B 0,C 180,E1 -27578.491,E2 -27578.491} C_VEL
LIN {X 0,Y 77.14,Z 369.767,A -85,B 0,C 180,E1 -27586.789,E2 -27586.789} C_VEL
LIN {X 0,Y 76.851,Z 365.652,A -85,B 0,C 180,E1 -27596.723,E2 -27596.723} C_VEL
LIN {X 0,Y 77.892,Z 361.242,A -85,B 0,C 180,E1 -27604.457,E2 -27604.457} C_VEL
LIN {X 0,Y 79.835,Z 355.918,A -85,B 0,C 180,E1 -27611.619,E2 -27611.619} C_VEL
LIN {X 0,Y 82.97,Z 348.7,A -85,B 0,C 180,E1 -27619.013,E2 -27619.013} C_VEL
LIN {X 0,Y 86.856,Z 340.36,A -85,B 0,C 180,E1 -27625.359,E2 -27625.359} C_VEL
LIN {X 0,Y 91.374,Z 330.473,A -85,B 0,C 180,E1 -27630.91,E2 -27630.91} C_VEL
LIN {X 0,Y 95.731,Z 320.052,A -85,B 0,C 180,E1 -27635.265,E2 -27635.265} C_VEL
LIN {X 0,Y 99.814,Z 308.992,A -85,B 0,C 180,E1 -27638.662,E2 -27638.662} C_VEL
LIN {X 0,Y 103.693,Z 296.441,A -85,B 0,C 180,E1 -27641.484,E2 -27641.484} C_VEL
LIN {X 0,Y 106.734,Z 283.479,A -85,B 0,C 180,E1 -27643.567,E2 -27643.567} C_VEL
LIN {X 0,Y 109.096,Z 269.3,A -85,B 0,C 180,E1 -27645.049,E2 -27645.049} C_VEL
LIN {X 0,Y 112.7,Z 232.887,A -85,B 0,C 180,E1 -27647.208,E2 -27647.208} C_VEL
LIN {X 0,Y 110.869,Z 228.252,A -85,B 0,C 180,E1 -27648.518,E2 -27648.518} C_VEL
LIN {X 0,Y 105.116,Z 216.177,A -85,B 0,C 180,E1 -27652.872,E2 -27652.872} C_VEL
LIN {X 0,Y 99.103,Z 205.699,A -85,B 0,C 180,E1 -27658.003,E2 -27658.003} C_VEL
LIN {X 0,Y 94.416,Z 198.479,A -85,B 0,C 180,E1 -27662.79,E2 -27662.79} C_VEL
LIN {X 0,Y 91.831,Z 194.715,A -85,B 0,C 180,E1 -27665.796,E2 -27665.796} C_VEL
LIN {X 0,Y 88.863,Z 191.027,A -85,B 0,C 180,E1 -27669.694,E2 -27669.694} C_VEL
LIN {X 0,Y 87.997,Z 189.581,A -85,B 0,C 180,E1 -27671.059,E2 -27671.059} C_VEL
LIN {X 0,Y 85.346,Z 186.922,A -85,B 0,C 180,E1 -27675.372,E2 -27675.372} C_VEL
LIN {X 0,Y 84.12,Z 184.375,A -85,B 0,C 180,E1 -27678.059,E2 -27678.059} C_VEL
LIN {X 0,Y 81.438,Z 182.673,A -85,B 0,C 180,E1 -27684.301,E2 -27684.301} C_VEL
LIN {X 0,Y 79.829,Z 180.198,A -85,B 0,C 180,E1 -27690.663,E2 -27690.663} C_VEL
LIN {X 0,Y 79.542,Z 178.556,A -85,B 0,C 180,E1 -27693.505,E2 -27693.505} C_VEL
LIN {X 0,Y 79.514,Z 178.559,A -85,B 0,C 180,E1 -27699.297,E2 -27699.297} C_VEL
LIN {X 0,Y 79.841,Z 178.523,A -85,B 0,C 180,E1 -27705.527,E2 -27705.527} C_VEL
LIN {X 0,Y 80.061,Z 178.562,A -85,B 0,C 180,E1 -27711.323,E2 -27711.323} C_VEL
LIN {X 0,Y 80.694,Z 180.485,A -85,B 0,C 180,E1 -27714.691,E2 -27714.691} C_VEL
LIN {X 0,Y 83.01,Z 183.064,A -85,B 0,C 180,E1 -27721.517,E2 -27721.517} C_VEL
LIN {X 0,Y 85.054,Z 184.67,A -85,B 0,C 180,E1 -27725.662,E2 -27725.662} C_VEL
LIN {X 0,Y 86.482,Z 187.585,A -85,B 0,C 180,E1 -27728.545,E2 -27728.545} C_VEL
LIN {X 0,Y 88.584,Z 189.771,A -85,B 0,C 180,E1 -27731.792,E2 -27731.792} C_VEL
LIN {X 0,Y 90.716,Z 193.304,A -85,B 0,C 180,E1 -27734.871,E2 -27734.871} C_VEL
LIN {X 0,Y 92.207,Z 195.063,A -85,B 0,C 180,E1 -27736.68,E2 -27736.68} C_VEL
LIN {X 0,Y 95.132,Z 199.695,A -85,B 0,C 180,E1 -27740.127,E2 -27740.127} C_VEL
LIN {X 0,Y 99.324,Z 206.261,A -85,B 0,C 180,E1 -27744.299,E2 -27744.299} C_VEL
LIN {X 0,Y 103.767,Z 214.502,A -85,B 0,C 180,E1 -27748.216,E2 -27748.216} C_VEL
LIN {X 0,Y 108.019,Z 226.424,A -85,B 0,C 180,E1 -27751.949,E2 -27751.949} C_VEL
LIN {X 0,Y 111.471,Z 237.97,A -85,B 0,C 180,E1 -27754.808,E2 -27754.808} C_VEL
LIN {X 0,Y 111.72,Z 247.34,A -85,B 0,C 180,E1 -27755.847,E2 -27755.847} C_VEL
LIN {X 0,Y 108.519,Z 279.232,A -85,B 0,C 180,E1 -27757.771,E2 -27757.771} C_VEL
LIN {X 0,Y 106.295,Z 291.83,A -85,B 0,C 180,E1 -27759.024,E2 -27759.024} C_VEL
LIN {X 0,Y 103.034,Z 305.058,A -85,B 0,C 180,E1 -27761.011,E2 -27761.011} C_VEL
LIN {X 0,Y 99.307,Z 316.632,A -85,B 0,C 180,E1 -27763.498,E2 -27763.498} C_VEL
LIN {X 0,Y 95.019,Z 327.903,A -85,B 0,C 180,E1 -27766.83,E2 -27766.83} C_VEL
LIN {X 0,Y 90.858,Z 337.546,A -85,B 0,C 180,E1 -27770.672,E2 -27770.672} C_VEL
LIN {X 0,Y 86.727,Z 346.496,A -85,B 0,C 180,E1 -27775.441,E2 -27775.441} C_VEL
LIN {X 0,Y 82.62,Z 355.628,A -85,B 0,C 180,E1 -27782.105,E2 -27782.105} C_VEL
LIN {X 0,Y 79.575,Z 362.937,A -85,B 0,C 180,E1 -27789.312,E2 -27789.312} C_VEL
LIN {X 0,Y 77.818,Z 368.753,A -85,B 0,C 180,E1 -27796.951,E2 -27796.951} C_VEL
LIN {X 0,Y 77.404,Z 373.285,A -85,B 0,C 180,E1 -27804.79,E2 -27804.79} C_VEL
LIN {X 0,Y 77.6,Z 375.613,A -85,B 0,C 180,E1 -27810,E2 -27810} C_VEL
LIN {X 0,Y 77.309,Z 377.378,A -85,B 0,C 180,E1 -27815.216,E2 -27815.216} C_VEL
LIN {X 0,Y 78.108,Z 379.687,A -85,B 0,C 180,E1 -27825.66,E2 -27825.66} C_VEL
LIN {X 0,Y 81.351,Z 380.452,A -85,B 0,C 180,E1 -27835.591,E2 -27835.591} C_VEL
LIN {X 0,Y 87.062,Z 379.814,A -85,B 0,C 180,E1 -27844.406,E2 -27844.406} C_VEL
LIN {X 0,Y 94.619,Z 377.722,A -85,B 0,C 180,E1 -27851.95,E2 -27851.95} C_VEL
LIN {X 0,Y 103.659,Z 374.094,A -85,B 0,C 180,E1 -27858.227,E2 -27858.227} C_VEL
LIN {X 0,Y 111.242,Z 370.309,A -85,B 0,C 180,E1 -27862.159,E2 -27862.159} C_VEL
LIN {X 0,Y 119.413,Z 365.49,A -85,B 0,C 180,E1 -27865.483,E2 -27865.483} C_VEL
LIN {X 0,Y 126.48,Z 360.624,A -85,B 0,C 180,E1 -27867.927,E2 -27867.927} C_VEL
LIN {X 0,Y 135.328,Z 353.544,A -85,B 0,C 180,E1 -27870.444,E2 -27870.444} C_VEL
LIN {X 0,Y 144.478,Z 344.858,A -85,B 0,C 180,E1 -27872.591,E2 -27872.591} C_VEL
LIN {X 0,Y 152.269,Z 336.064,A -85,B 0,C 180,E1 -27874.161,E2 -27874.161} C_VEL
LIN {X 0,Y 160.201,Z 325.34,A -85,B 0,C 180,E1 -27875.546,E2 -27875.546} C_VEL
LIN {X 0,Y 167.518,Z 313.074,A -85,B 0,C 180,E1 -27876.596,E2 -27876.596} C_VEL
LIN {X 0,Y 172.913,Z 301.706,A -85,B 0,C 180,E1 -27877.304,E2 -27877.304} C_VEL
LIN {X 0,Y 177.619,Z 288.73,A -85,B 0,C 180,E1 -27877.901,E2 -27877.901} C_VEL
LIN {X 0,Y 178.822,Z 284.605,A -85,B 0,C 180,E1 -27878.103,E2 -27878.103} C_VEL
LIN {X 0,Y 178.894,Z 282.866,A -85,B 0,C 180,E1 -27879.92,E2 -27879.92} C_VEL
LIN {X 0,Y 178.903,Z 282.058,A -85,B 0,C 180,E1 -27881.683,E2 -27881.683} C_VEL
LIN {X 0,Y 178.916,Z 282.049,A -85,B 0,C 180,E1 -27882.706,E2 -27882.706} C_VEL
LIN {X 0,Y 178.734,Z 282.856,A -85,B 0,C 180,E1 -27883.385,E2 -27883.385} C_VEL
LIN {X 0,Y 178.286,Z 284.605,A -85,B 0,C 180,E1 -27883.887,E2 -27883.887} C_VEL
LIN {X 0,Y 177.273,Z 288.113,A -85,B 0,C 180,E1 -27884.337,E2 -27884.337} C_VEL
LIN {X 0,Y 174.658,Z 295.467,A -85,B 0,C 180,E1 -27884.43,E2 -27884.43} C_VEL
LIN {X 0,Y 172.161,Z 301.438,A -85,B 0,C 180,E1 -27884.557,E2 -27884.557} C_VEL
LIN {X 0,Y 166.431,Z 312.927,A -85,B 0,C 180,E1 -27885.494,E2 -27885.494} C_VEL
LIN {X 0,Y 159.827,Z 323.519,A -85,B 0,C 180,E1 -27886.627,E2 -27886.627} C_VEL
LIN {X 0,Y 151.688,Z 334.04,A -85,B 0,C 180,E1 -27888.142,E2 -27888.142} C_VEL
LIN {X 0,Y 144.261,Z 342.048,A -85,B 0,C 180,E1 -27889.677,E2 -27889.677} C_VEL
LIN {X 0,Y 134.86,Z 350.548,A -85,B 0,C 180,E1 -27891.95,E2 -27891.95} C_VEL
LIN {X 0,Y 125.287,Z 357.637,A -85,B 0,C 180,E1 -27894.672,E2 -27894.672} C_VEL
LIN {X 0,Y 115.827,Z 363.311,A -85,B 0,C 180,E1 -27897.851,E2 -27897.851} C_VEL
LIN {X 0,Y 105.502,Z 368.243,A -85,B 0,C 180,E1 -27902.279,E2 -27902.279} C_VEL
LIN {X 0,Y 98.907,Z 370.702,A -85,B 0,C 180,E1 -27905.856,E2 -27905.856} C_VEL
LIN {X 0,Y 92.732,Z 372.506,A -85,B 0,C 180,E1 -27909.859,E2 -27909.859} C_VEL
LIN {X 0,Y 87.095,Z 373.609,A -85,B 0,C 180,E1 -27914.463,E2 -27914.463} C_VEL
LIN {X 0,Y 81.623,Z 374.13,A -85,B 0,C 180,E1 -27920.145,E2 -27920.145} C_VEL
LIN {X 0,Y 76.618,Z 373.836,A -85,B 0,C 180,E1 -27927.298,E2 -27927.298} C_VEL
LIN {X 0,Y 72.77,Z 372.582,A -85,B 0,C 180,E1 -27935.412,E2 -27935.412} C_VEL
LIN {X 0,Y 70.195,Z 369.913,A -85,B 0,C 180,E1 -27945.506,E2 -27945.506} C_VEL
LIN {X 0,Y 69.625,Z 366.84,A -85,B 0,C 180,E1 -27953.853,E2 -27953.853} C_VEL
LIN {X 0,Y 70.576,Z 361.953,A -85,B 0,C 180,E1 -27963.664,E2 -27963.664} C_VEL
LIN {X 0,Y 72.539,Z 356.661,A -85,B 0,C 180,E1 -27971.647,E2 -27971.647} C_VEL
LIN {X 0,Y 76.148,Z 348.817,A -85,B 0,C 180,E1 -27980.454,E2 -27980.454} C_VEL
LIN {X 0,Y 80.504,Z 340.035,A -85,B 0,C 180,E1 -27987.498,E2 -27987.498} C_VEL
LIN {X 0,Y 85.037,Z 330.641,A -85,B 0,C 180,E1 -27993.021,E2 -27993.021} C_VEL
LIN {X 0,Y 89.419,Z 320.768,A -85,B 0,C 180,E1 -27997.338,E2 -27997.338} C_VEL
LIN {X 0,Y 94.002,Z 309.015,A -85,B 0,C 180,E1 -28001.076,E2 -28001.076} C_VEL
LIN {X 0,Y 98.14,Z 296.244,A -85,B 0,C 180,E1 -28003.986,E2 -28003.986} C_VEL
LIN {X 0,Y 101.19,Z 283.793,A -85,B 0,C 180,E1 -28006,E2 -28006} C_VEL
LIN {X 0,Y 103.615,Z 269.91,A -85,B 0,C 180,E1 -28007.481,E2 -28007.481} C_VEL
LIN {X 0,Y 107.288,Z 234.772,A -85,B 0,C 180,E1 -28009.596,E2 -28009.596} C_VEL
LIN {X 0,Y 101.317,Z 221.463,A -85,B 0,C 180,E1 -28014.503,E2 -28014.503} C_VEL
LIN {X 0,Y 95.484,Z 210.819,A -85,B 0,C 180,E1 -28020.015,E2 -28020.015} C_VEL
LIN {X 0,Y 91.582,Z 204.447,A -85,B 0,C 180,E1 -28024.394,E2 -28024.394} C_VEL
LIN {X 0,Y 88.496,Z 200.054,A -85,B 0,C 180,E1 -28028.354,E2 -28028.354} C_VEL
LIN {X 0,Y 86.07,Z 196.422,A -85,B 0,C 180,E1 -28032.12,E2 -28032.12} C_VEL
LIN {X 0,Y 82.921,Z 192.587,A -85,B 0,C 180,E1 -28037.883,E2 -28037.883} C_VEL
LIN {X 0,Y 82.338,Z 191.188,A -85,B 0,C 180,E1 -28039.367,E2 -28039.367} C_VEL
LIN {X 0,Y 79.457,Z 188.759,A -85,B 0,C 180,E1 -28047.377,E2 -28047.377} C_VEL
LIN {X 0,Y 78.406,Z 186.398,A -85,B 0,C 180,E1 -28053.09,E2 -28053.09} C_VEL
LIN {X 0,Y 78.292,Z 185.559,A -85,B 0,C 180,E1 -28054.619,E2 -28054.619} C_VEL
LIN {X 0,Y 78.756,Z 185.502,A -85,B 0,C 180,E1 -28070.045,E2 -28070.045} C_VEL
LIN {X 0,Y 79.592,Z 187.678,A -85,B 0,C 180,E1 -28074.618,E2 -28074.618} C_VEL
LIN {X 0,Y 83.014,Z 191.241,A -85,B 0,C 180,E1 -28083.945,E2 -28083.945} C_VEL
LIN {X 0,Y 84.724,Z 194.409,A -85,B 0,C 180,E1 -28087.568,E2 -28087.568} C_VEL
LIN {X 0,Y 86.265,Z 196.203,A -85,B 0,C 180,E1 -28090.19,E2 -28090.19} C_VEL
LIN {X 0,Y 88.58,Z 199.886,A -85,B 0,C 180,E1 -28093.771,E2 -28093.771} C_VEL
LIN {X 0,Y 91.442,Z 204.169,A -85,B 0,C 180,E1 -28097.472,E2 -28097.472} C_VEL
LIN {X 0,Y 95.682,Z 211.337,A -85,B 0,C 180,E1 -28102.297,E2 -28102.297} C_VEL
LIN {X 0,Y 99.626,Z 219.011,A -85,B 0,C 180,E1 -28106.162,E2 -28106.162} C_VEL
LIN {X 0,Y 103.486,Z 230.539,A -85,B 0,C 180,E1 -28109.952,E2 -28109.952} C_VEL
LIN {X 0,Y 106.22,Z 240.17,A -85,B 0,C 180,E1 -28112.52,E2 -28112.52} C_VEL
LIN {X 0,Y 106.312,Z 248.2,A -85,B 0,C 180,E1 -28113.435,E2 -28113.435} C_VEL
LIN {X 0,Y 103.077,Z 278.829,A -85,B 0,C 180,E1 -28115.309,E2 -28115.309} C_VEL
LIN {X 0,Y 100.699,Z 291.748,A -85,B 0,C 180,E1 -28116.62,E2 -28116.62} C_VEL
LIN {X 0,Y 97.611,Z 303.867,A -85,B 0,C 180,E1 -28118.464,E2 -28118.464} C_VEL
LIN {X 0,Y 93.381,Z 316.406,A -85,B 0,C 180,E1 -28121.183,E2 -28121.183} C_VEL
LIN {X 0,Y 88.879,Z 327.652,A -85,B 0,C 180,E1 -28124.63,E2 -28124.63} C_VEL
LIN {X 0,Y 83.994,Z 338.296,A -85,B 0,C 180,E1 -28129.154,E2 -28129.154} C_VEL
LIN {X 0,Y 79.284,Z 347.831,A -85,B 0,C 180,E1 -28134.817,E2 -28134.817} C_VEL
LIN {X 0,Y 75.1,Z 356.663,A -85,B 0,C 180,E1 -28142.101,E2 -28142.101} C_VEL
LIN {X 0,Y 72.098,Z 363.649,A -85,B 0,C 180,E1 -28150.052,E2 -28150.052} C_VEL
LIN {X 0,Y 70.554,Z 369.213,A -85,B 0,C 180,E1 -28158.508,E2 -28158.508} C_VEL
LIN {X 0,Y 70.388,Z 373.402,A -85,B 0,C 180,E1 -28166.846,E2 -28166.846} C_VEL
LIN {X 0,Y 70.538,Z 374.715,A -85,B 0,C 180,E1 -28170,E2 -28170} C_VEL
LIN {X 0,Y 70.253,Z 376.548,A -85,B 0,C 180,E1 -28175.741,E2 -28175.741} C_VEL
LIN {X 0,Y 71.278,Z 379.011,A -85,B 0,C 180,E1 -28187.205,E2 -28187.205} C_VEL
LIN {X 0,Y 74.986,Z 380.015,A -85,B 0,C 180,E1 -28197.944,E2 -28197.944} C_VEL
LIN {X 0,Y 81.284,Z 379.546,A -85,B 0,C 180,E1 -28207.245,E2 -28207.245} C_VEL
LIN {X 0,Y 89.452,Z 377.666,A -85,B 0,C 180,E1 -28214.999,E2 -28214.999} C_VEL
LIN {X 0,Y 94.118,Z 376.184,A -85,B 0,C 180,E1 -28218.307,E2 -28218.307} C_VEL
LIN {X 0,Y 101.66,Z 373.189,A -85,B 0,C 180,E1 -28222.657,E2 -28222.657} C_VEL
LIN {X 0,Y 109.83,Z 369.257,A -85,B 0,C 180,E1 -28226.29,E2 -28226.29} C_VEL
LIN {X 0,Y 118.429,Z 364.322,A -85,B 0,C 180,E1 -28229.37,E2 -28229.37} C_VEL
LIN {X 0,Y 128.973,Z 357.075,A -85,B 0,C 180,E1 -28232.312,E2 -28232.312} C_VEL
LIN {X 0,Y 138.241,Z 349.292,A -85,B 0,C 180,E1 -28234.472,E2 -28234.472} C_VEL
LIN {X 0,Y 147.752,Z 339.712,A -85,B 0,C 180,E1 -28236.297,E2 -28236.297} C_VEL
LIN {X 0,Y 155.836,Z 329.958,A -85,B 0,C 180,E1 -28237.595,E2 -28237.595} C_VEL
LIN {X 0,Y 163.233,Z 319.089,A -85,B 0,C 180,E1 -28238.6,E2 -28238.6} C_VEL
LIN {X 0,Y 169.685,Z 307.348,A -85,B 0,C 180,E1 -28239.366,E2 -28239.366} C_VEL
LIN {X 0,Y 174.828,Z 295.419,A -85,B 0,C 180,E1 -28239.944,E2 -28239.944} C_VEL
LIN {X 0,Y 176.469,Z 290.741,A -85,B 0,C 180,E1 -28240.127,E2 -28240.127} C_VEL
LIN {X 0,Y 176.875,Z 289.188,A -85,B 0,C 180,E1 -28240.986,E2 -28240.986} C_VEL
LIN {X 0,Y 176.882,Z 288.849,A -85,B 0,C 180,E1 -28242.473,E2 -28242.473} C_VEL
LIN {X 0,Y 176.726,Z 289.587,A -85,B 0,C 180,E1 -28243.836,E2 -28243.836} C_VEL
LIN {X 0,Y 172.161,Z 301.438,A -85,B 0,C 180,E1 -28244.557,E2 -28244.557} C_VEL
LIN {X 0,Y 170.464,Z 305.125,A -85,B 0,C 180,E1 -28244.584,E2 -28244.584} C_VEL
LIN {X 0,Y 164.07,Z 316.641,A -85,B 0,C 180,E1 -28243.553,E2 -28243.553} C_VEL
LIN {X 0,Y 161.977,Z 319.951,A -85,B 0,C 180,E1 -28243.637,E2 -28243.637} C_VEL
LIN {X 0,Y 153.73,Z 331.174,A -85,B 0,C 180,E1 -28244.951,E2 -28244.951} C_VEL
LIN {X 0,Y 145.857,Z 339.955,A -85,B 0,C 180,E1 -28246.315,E2 -28246.315} C_VEL
LIN {X 0,Y 136.387,Z 348.689,A -85,B 0,C 180,E1 -28248.253,E2 -28248.253} C_VEL
LIN {X 0,Y 127.093,Z 355.716,A -85,B 0,C 180,E1 -28250.45,E2 -28250.45} C_VEL
LIN {X 0,Y 117.529,Z 361.7,A -85,B 0,C 180,E1 -28253.13,E2 -28253.13} C_VEL
LIN {X 0,Y 108.276,Z 366.392,A -85,B 0,C 180,E1 -28256.278,E2 -28256.278} C_VEL
LIN {X 0,Y 98.395,Z 370.304,A -85,B 0,C 180,E1 -28260.528,E2 -28260.528} C_VEL
LIN {X 0,Y 91.335,Z 372.382,A -85,B 0,C 180,E1 -28264.412,E2 -28264.412} C_VEL
LIN {X 0,Y 83.73,Z 373.931,A -85,B 0,C 180,E1 -28269.663,E2 -28269.663} C_VEL
LIN {X 0,Y 76.99,Z 374.559,A -85,B 0,C 180,E1 -28275.893,E2 -28275.893} C_VEL
LIN {X 0,Y 69.977,Z 374.031,A -85,B 0,C 180,E1 -28285.327,E2 -28285.327} C_VEL
LIN {X 0,Y 66.519,Z 372.935,A -85,B 0,C 180,E1 -28292.305,E2 -28292.305} C_VEL
LIN {X 0,Y 63.751,Z 370.805,A -85,B 0,C 180,E1 -28301.408,E2 -28301.408} C_VEL
LIN {X 0,Y 62.548,Z 367.419,A -85,B 0,C 180,E1 -28311.86,E2 -28311.86} C_VEL
LIN {X 0,Y 63.393,Z 362.126,A -85,B 0,C 180,E1 -28323.676,E2 -28323.676} C_VEL
LIN {X 0,Y 65.891,Z 355.936,A -85,B 0,C 180,E1 -28333.725,E2 -28333.725} C_VEL
LIN {X 0,Y 69.72,Z 348.226,A -85,B 0,C 180,E1 -28342.762,E2 -28342.762} C_VEL
LIN {X 0,Y 74.264,Z 339.611,A -85,B 0,C 180,E1 -28350,E2 -28350} C_VEL
LIN {X 0,Y 79.115,Z 330.191,A -85,B 0,C 180,E1 -28355.736,E2 -28355.736} C_VEL
LIN {X 0,Y 84.102,Z 319.488,A -85,B 0,C 180,E1 -28360.43,E2 -28360.43} C_VEL
LIN {X 0,Y 89.019,Z 307.201,A -85,B 0,C 180,E1 -28364.283,E2 -28364.283} C_VEL
LIN {X 0,Y 93.156,Z 294.722,A -85,B 0,C 180,E1 -28366.998,E2 -28366.998} C_VEL
LIN {X 0,Y 96.522,Z 280.864,A -85,B 0,C 180,E1 -28369.124,E2 -28369.124} C_VEL
LIN {X 0,Y 98.634,Z 268.332,A -85,B 0,C 180,E1 -28370.355,E2 -28370.355} C_VEL
LIN {X 0,Y 102.032,Z 236.93,A -85,B 0,C 180,E1 -28372.227,E2 -28372.227} C_VEL
LIN {X 0,Y 96.951,Z 225.421,A -85,B 0,C 180,E1 -28376.866,E2 -28376.866} C_VEL
LIN {X 0,Y 91.963,Z 215.865,A -85,B 0,C 180,E1 -28382.212,E2 -28382.212} C_VEL
LIN {X 0,Y 88.147,Z 209.584,A -85,B 0,C 180,E1 -28386.945,E2 -28386.945} C_VEL
LIN {X 0,Y 85.859,Z 206.001,A -85,B 0,C 180,E1 -28390.32,E2 -28390.32} C_VEL
LIN {X 0,Y 83.411,Z 202.217,A -85,B 0,C 180,E1 -28394.582,E2 -28394.582} C_VEL
LIN {X 0,Y 80.872,Z 198.718,A -85,B 0,C 180,E1 -28399.937,E2 -28399.937} C_VEL
LIN {X 0,Y 80.321,Z 197.727,A -85,B 0,C 180,E1 -28401.433,E2 -28401.433} C_VEL
LIN {X 0,Y 77.452,Z 194.385,A -85,B 0,C 180,E1 -28411.851,E2 -28411.851} C_VEL
LIN {X 0,Y 77.127,Z 192.558,A -85,B 0,C 180,E1 -28415.675,E2 -28415.675} C_VEL
LIN {X 0,Y 77.488,Z 192.485,A -85,B 0,C 180,E1 -28428.835,E2 -28428.835} C_VEL
LIN {X 0,Y 78.922,Z 195.388,A -85,B 0,C 180,E1 -28436.172,E2 -28436.172} C_VEL
LIN {X 0,Y 81.111,Z 197.845,A -85,B 0,C 180,E1 -28442.329,E2 -28442.329} C_VEL
LIN {X 0,Y 83.117,Z 201.297,A -85,B 0,C 180,E1 -28446.79,E2 -28446.79} C_VEL
LIN {X 0,Y 84.118,Z 202.801,A -85,B 0,C 180,E1 -28448.691,E2 -28448.691} C_VEL
LIN {X 0,Y 87.368,Z 208.042,A -85,B 0,C 180,E1 -28453.966,E2 -28453.966} C_VEL
LIN {X 0,Y 92.059,Z 216.157,A -85,B 0,C 180,E1 -28460.008,E2 -28460.008} C_VEL
LIN {X 0,Y 95.637,Z 223.646,A -85,B 0,C 180,E1 -28464.009,E2 -28464.009} C_VEL
LIN {X 0,Y 99.413,Z 235.831,A -85,B 0,C 180,E1 -28468.144,E2 -28468.144} C_VEL
LIN {X 0,Y 101.181,Z 243.031,A -85,B 0,C 180,E1 -28470.094,E2 -28470.094} C_VEL
LIN {X 0,Y 101.011,Z 250.013,A -85,B 0,C 180,E1 -28470.825,E2 -28470.825} C_VEL
LIN {X 0,Y 97.842,Z 278.531,A -85,B 0,C 180,E1 -28472.593,E2 -28472.593} C_VEL
LIN {X 0,Y 95.301,Z 291.689,A -85,B 0,C 180,E1 -28473.944,E2 -28473.944} C_VEL
LIN {X 0,Y 92.06,Z 303.7,A -85,B 0,C 180,E1 -28475.794,E2 -28475.794} C_VEL
LIN {X 0,Y 87.634,Z 316.185,A -85,B 0,C 180,E1 -28478.563,E2 -28478.563} C_VEL
LIN {X 0,Y 82.787,Z 327.664,A -85,B 0,C 180,E1 -28482.21,E2 -28482.21} C_VEL
LIN {X 0,Y 77.737,Z 337.978,A -85,B 0,C 180,E1 -28486.809,E2 -28486.809} C_VEL
LIN {X 0,Y 72.7,Z 347.503,A -85,B 0,C 180,E1 -28492.829,E2 -28492.829} C_VEL
LIN {X 0,Y 68.223,Z 356.304,A -85,B 0,C 180,E1 -28500.704,E2 -28500.704} C_VEL
LIN {X 0,Y 65.059,Z 363.271,A -85,B 0,C 180,E1 -28509.446,E2 -28509.446} C_VEL
LIN {X 0,Y 63.378,Z 369.622,A -85,B 0,C 180,E1 -28520.425,E2 -28520.425} C_VEL
LIN {X 0,Y 63.47,Z 373.705,A -85,B 0,C 180,E1 -28530,E2 -28530} C_VEL
LIN {X 0,Y 63.225,Z 375.687,A -85,B 0,C 180,E1 -28536.382,E2 -28536.382} C_VEL
LIN {X 0,Y 64.522,Z 378.329,A -85,B 0,C 180,E1 -28549.072,E2 -28549.072} C_VEL
LIN {X 0,Y 68.776,Z 379.506,A -85,B 0,C 180,E1 -28560.726,E2 -28560.726} C_VEL
LIN {X 0,Y 75.738,Z 379.284,A -85,B 0,C 180,E1 -28570.507,E2 -28570.507} C_VEL
LIN {X 0,Y 84.574,Z 377.584,A -85,B 0,C 180,E1 -28578.407,E2 -28578.407} C_VEL
LIN {X 0,Y 94.785,Z 374.445,A -85,B 0,C 180,E1 -28584.647,E2 -28584.647} C_VEL
LIN {X 0,Y 103.167,Z 371.044,A -85,B 0,C 180,E1 -28588.378,E2 -28588.378} C_VEL
LIN {X 0,Y 112.016,Z 366.666,A -85,B 0,C 180,E1 -28591.446,E2 -28591.446} C_VEL
LIN {X 0,Y 121.156,Z 361.204,A -85,B 0,C 180,E1 -28594.042,E2 -28594.042} C_VEL
LIN {X 0,Y 130.567,Z 354.487,A -85,B 0,C 180,E1 -28596.213,E2 -28596.213} C_VEL
LIN {X 0,Y 140.213,Z 346.3,A -85,B 0,C 180,E1 -28598.014,E2 -28598.014} C_VEL
LIN {X 0,Y 148.376,Z 338.004,A -85,B 0,C 180,E1 -28599.305,E2 -28599.305} C_VEL
LIN {X 0,Y 156.633,Z 327.912,A -85,B 0,C 180,E1 -28600.432,E2 -28600.432} C_VEL
LIN {X 0,Y 164.19,Z 316.65,A -85,B 0,C 180,E1 -28601.268,E2 -28601.268} C_VEL
LIN {X 0,Y 170.111,Z 305.71,A -85,B 0,C 180,E1 -28601.845,E2 -28601.845} C_VEL
LIN {X 0,Y 170.963,Z 303.816,A -85,B 0,C 180,E1 -28602.313,E2 -28602.313} C_VEL
LIN {X 0,Y 164.598,Z 315.761,A -85,B 0,C 180,E1 -28603.246,E2 -28603.246} C_VEL
LIN {X 0,Y 161.977,Z 319.951,A -85,B 0,C 180,E1 -28603.637,E2 -28603.637} C_VEL
LIN {X 0,Y 158.671,Z 324.806,A -85,B 0,C 180,E1 -28603.908,E2 -28603.908} C_VEL
LIN {X 0,Y 149.901,Z 335.584,A -85,B 0,C 180,E1 -28603.654,E2 -28603.654} C_VEL
LIN {X 0,Y 144.439,Z 341.299,A -85,B 0,C 180,E1 -28603.748,E2 -28603.748} C_VEL
LIN {X 0,Y 141.677,Z 343.888,A -85,B 0,C 180,E1 -28604.091,E2 -28604.091} C_VEL
LIN {X 0,Y 132.177,Z 351.837,A -85,B 0,C 180,E1 -28605.867,E2 -28605.867} C_VEL
LIN {X 0,Y 122.108,Z 358.694,A -85,B 0,C 180,E1 -28608.08,E2 -28608.08} C_VEL
LIN {X 0,Y 114.136,Z 363.196,A -85,B 0,C 180,E1 -28610.131,E2 -28610.131} C_VEL
LIN {X 0,Y 102.501,Z 368.428,A -85,B 0,C 180,E1 -28613.821,E2 -28613.821} C_VEL
LIN {X 0,Y 91.393,Z 372.093,A -85,B 0,C 180,E1 -28618.537,E2 -28618.537} C_VEL
LIN {X 0,Y 80.243,Z 374.361,A -85,B 0,C 180,E1 -28625.024,E2 -28625.024} C_VEL
LIN {X 0,Y 71.864,Z 374.993,A -85,B 0,C 180,E1 -28632.056,E2 -28632.056} C_VEL
LIN {X 0,Y 66.323,Z 374.718,A -85,B 0,C 180,E1 -28638.534,E2 -28638.534} C_VEL
LIN {X 0,Y 61.063,Z 373.504,A -85,B 0,C 180,E1 -28647.41,E2 -28647.41} C_VEL
LIN {X 0,Y 57.314,Z 371.279,A -85,B 0,C 180,E1 -28657.813,E2 -28657.813} C_VEL
LIN {X 0,Y 55.492,Z 367.488,A -85,B 0,C 180,E1 -28670.71,E2 -28670.71} C_VEL
LIN {X 0,Y 55.938,Z 363.264,A -85,B 0,C 180,E1 -28681.576,E2 -28681.576} C_VEL
LIN {X 0,Y 57.862,Z 358.262,A -85,B 0,C 180,E1 -28691.375,E2 -28691.375} C_VEL
LIN {X 0,Y 61.496,Z 350.98,A -85,B 0,C 180,E1 -28701.787,E2 -28701.787} C_VEL
LIN {X 0,Y 66.033,Z 342.911,A -85,B 0,C 180,E1 -28710,E2 -28710} C_VEL
LIN {X 0,Y 70.669,Z 334.678,A -85,B 0,C 180,E1 -28716.028,E2 -28716.028} C_VEL
LIN {X 0,Y 75.927,Z 324.654,A -85,B 0,C 180,E1 -28721.301,E2 -28721.301} C_VEL
LIN {X 0,Y 81.343,Z 312.874,A -85,B 0,C 180,E1 -28725.664,E2 -28725.664} C_VEL
LIN {X 0,Y 85.919,Z 300.912,A -85,B 0,C 180,E1 -28728.789,E2 -28728.789} C_VEL
LIN {X 0,Y 89.711,Z 288.12,A -85,B 0,C 180,E1 -28731.139,E2 -28731.139} C_VEL
LIN {X 0,Y 92.65,Z 274.618,A -85,B 0,C 180,E1 -28732.8,E2 -28732.8} C_VEL
LIN {X 0,Y 94.764,Z 258.655,A -85,B 0,C 180,E1 -28733.938,E2 -28733.938} C_VEL
LIN {X 0,Y 96.873,Z 239.402,A -85,B 0,C 180,E1 -28735.069,E2 -28735.069} C_VEL
LIN {X 0,Y 93.029,Z 230.01,A -85,B 0,C 180,E1 -28739.144,E2 -28739.144} C_VEL
LIN {X 0,Y 88.588,Z 221.068,A -85,B 0,C 180,E1 -28744.447,E2 -28744.447} C_VEL
LIN {X 0,Y 85.513,Z 215.531,A -85,B 0,C 180,E1 -28748.782,E2 -28748.782} C_VEL
LIN {X 0,Y 83.319,Z 211.867,A -85,B 0,C 180,E1 -28752.439,E2 -28752.439} C_VEL
LIN {X 0,Y 81.166,Z 208.408,A -85,B 0,C 180,E1 -28756.57,E2 -28756.57} C_VEL
LIN {X 0,Y 78.957,Z 204.903,A -85,B 0,C 180,E1 -28762.015,E2 -28762.015} C_VEL
LIN {X 0,Y 76.099,Z 200.675,A -85,B 0,C 180,E1 -28774.301,E2 -28774.301} C_VEL
LIN {X 0,Y 75.993,Z 199.557,A -85,B 0,C 180,E1 -28776.713,E2 -28776.713} C_VEL
LIN {X 0,Y 76.34,Z 199.614,A -85,B 0,C 180,E1 -28788.3,E2 -28788.3} C_VEL
LIN {X 0,Y 77.831,Z 202.484,A -85,B 0,C 180,E1 -28796.118,E2 -28796.118} C_VEL
LIN {X 0,Y 79.334,Z 204.532,A -85,B 0,C 180,E1 -28800.794,E2 -28800.794} C_VEL
LIN {X 0,Y 81.432,Z 208.117,A -85,B 0,C 180,E1 -28805.824,E2 -28805.824} C_VEL
LIN {X 0,Y 84.971,Z 214.361,A -85,B 0,C 180,E1 -28812.396,E2 -28812.396} C_VEL
LIN {X 0,Y 88.984,Z 221.937,A -85,B 0,C 180,E1 -28818.12,E2 -28818.12} C_VEL
LIN {X 0,Y 91.738,Z 228.118,A -85,B 0,C 180,E1 -28821.602,E2 -28821.602} C_VEL
LIN {X 0,Y 94.924,Z 239.444,A -85,B 0,C 180,E1 -28825.674,E2 -28825.674} C_VEL
LIN {X 0,Y 96.269,Z 244.985,A -85,B 0,C 180,E1 -28827.318,E2 -28827.318} C_VEL
LIN {X 0,Y 95.963,Z 251.349,A -85,B 0,C 180,E1 -28827.943,E2 -28827.943} C_VEL
LIN {X 0,Y 92.74,Z 278.581,A -85,B 0,C 180,E1 -28829.636,E2 -28829.636} C_VEL
LIN {X 0,Y 90.143,Z 291.342,A -85,B 0,C 180,E1 -28830.95,E2 -28830.95} C_VEL
LIN {X 0,Y 86.74,Z 303.325,A -85,B 0,C 180,E1 -28832.794,E2 -28832.794} C_VEL
LIN {X 0,Y 82.098,Z 315.786,A -85,B 0,C 180,E1 -28835.586,E2 -28835.586} C_VEL
LIN {X 0,Y 77.091,Z 326.98,A -85,B 0,C 180,E1 -28839.204,E2 -28839.204} C_VEL
LIN {X 0,Y 71.808,Z 337.182,A -85,B 0,C 180,E1 -28843.866,E2 -28843.866} C_VEL
LIN {X 0,Y 66.233,Z 347.078,A -85,B 0,C 180,E1 -28850.457,E2 -28850.457} C_VEL
LIN {X 0,Y 61.416,Z 355.886,A -85,B 0,C 180,E1 -28859.006,E2 -28859.006} C_VEL
LIN {X 0,Y 58.006,Z 362.851,A -85,B 0,C 180,E1 -28868.686,E2 -28868.686} C_VEL
LIN {X 0,Y 56.38,Z 368.399,A -85,B 0,C 180,E1 -28879.223,E2 -28879.223} C_VEL
LIN {X 0,Y 56.403,Z 372.68,A -85,B 0,C 180,E1 -28890,E2 -28890} C_VEL
LIN {X 0,Y 56.222,Z 374.756,A -85,B 0,C 180,E1 -28897.181,E2 -28897.181} C_VEL
LIN {X 0,Y 57.859,Z 377.629,A -85,B 0,C 180,E1 -28911.37,E2 -28911.37} C_VEL
LIN {X 0,Y 62.765,Z 378.98,A -85,B 0,C 180,E1 -28924.046,E2 -28924.046} C_VEL
LIN {X 0,Y 70.478,Z 378.949,A -85,B 0,C 180,E1 -28934.269,E2 -28934.269} C_VEL
LIN {X 0,Y 80.02,Z 377.512,A -85,B 0,C 180,E1 -28942.227,E2 -28942.227} C_VEL
LIN {X 0,Y 90.867,Z 374.582,A -85,B 0,C 180,E1 -28948.295,E2 -28948.295} C_VEL
LIN {X 0,Y 102.644,Z 370.121,A -85,B 0,C 180,E1 -28952.886,E2 -28952.886} C_VEL
LIN {X 0,Y 111.907,Z 365.62,A -85,B 0,C 180,E1 -28955.592,E2 -28955.592} C_VEL
LIN {X 0,Y 123.08,Z 358.986,A -85,B 0,C 180,E1 -28958.108,E2 -28958.108} C_VEL
LIN {X 0,Y 132.81,Z 351.886,A -85,B 0,C 180,E1 -28959.931,E2 -28959.931} C_VEL
LIN {X 0,Y 142.712,Z 343.172,A -85,B 0,C 180,E1 -28961.437,E2 -28961.437} C_VEL
LIN {X 0,Y 147.73,Z 338.076,A -85,B 0,C 180,E1 -28962.075,E2 -28962.075} C_VEL
LIN {X 0,Y 149.144,Z 336.441,A -85,B 0,C 180,E1 -28962.894,E2 -28962.894} C_VEL
LIN {X 0,Y 141.677,Z 343.888,A -85,B 0,C 180,E1 -28964.091,E2 -28964.091} C_VEL
LIN {X 0,Y 137.335,Z 347.733,A -85,B 0,C 180,E1 -28964.586,E2 -28964.586} C_VEL
LIN {X 0,Y 129.484,Z 353.79,A -85,B 0,C 180,E1 -28964.757,E2 -28964.757} C_VEL
LIN {X 0,Y 121.233,Z 359.22,A -85,B 0,C 180,E1 -28965.017,E2 -28965.017} C_VEL
LIN {X 0,Y 116.286,Z 362.007,A -85,B 0,C 180,E1 -28965.741,E2 -28965.741} C_VEL
LIN {X 0,Y 105.363,Z 367.174,A -85,B 0,C 180,E1 -28968.456,E2 -28968.456} C_VEL
LIN {X 0,Y 95.575,Z 370.737,A -85,B 0,C 180,E1 -28971.542,E2 -28971.542} C_VEL
LIN {X 0,Y 84.527,Z 373.611,A -85,B 0,C 180,E1 -28976.139,E2 -28976.139} C_VEL
LIN {X 0,Y 77.307,Z 374.798,A -85,B 0,C 180,E1 -28980.065,E2 -28980.065} C_VEL
LIN {X 0,Y 69.202,Z 375.422,A -85,B 0,C 180,E1 -28985.828,E2 -28985.828} C_VEL
LIN {X 0,Y 61.923,Z 375.153,A -85,B 0,C 180,E1 -28993.119,E2 -28993.119} C_VEL
LIN {X 0,Y 54.322,Z 373.421,A -85,B 0,C 180,E1 -29005.092,E2 -29005.092} C_VEL
LIN {X 0,Y 49.752,Z 370.386,A -85,B 0,C 180,E1 -29019.02,E2 -29019.02} C_VEL
LIN {X 0,Y 48.37,Z 365.866,A -85,B 0,C 180,E1 -29034.467,E2 -29034.467} C_VEL
LIN {X 0,Y 49.59,Z 360.935,A -85,B 0,C 180,E1 -29047.064,E2 -29047.064} C_VEL
LIN {X 0,Y 52.595,Z 354.873,A -85,B 0,C 180,E1 -29058.438,E2 -29058.438} C_VEL
LIN {X 0,Y 57.107,Z 347.233,A -85,B 0,C 180,E1 -29068.596,E2 -29068.596} C_VEL
LIN {X 0,Y 62.358,Z 338.68,A -85,B 0,C 180,E1 -29076.471,E2 -29076.471} C_VEL
LIN {X 0,Y 68.104,Z 328.821,A -85,B 0,C 180,E1 -29082.668,E2 -29082.668} C_VEL
LIN {X 0,Y 73.642,Z 318.056,A -85,B 0,C 180,E1 -29087.383,E2 -29087.383} C_VEL
LIN {X 0,Y 78.712,Z 306.49,A -85,B 0,C 180,E1 -29090.925,E2 -29090.925} C_VEL
LIN {X 0,Y 83.291,Z 293.525,A -85,B 0,C 180,E1 -29093.628,E2 -29093.628} C_VEL
LIN {X 0,Y 86.717,Z 280.293,A -85,B 0,C 180,E1 -29095.559,E2 -29095.559} C_VEL
LIN {X 0,Y 89.082,Z 266.638,A -85,B 0,C 180,E1 -29096.771,E2 -29096.771} C_VEL
LIN {X 0,Y 92.009,Z 241.725,A -85,B 0,C 180,E1 -29098.222,E2 -29098.222} C_VEL
LIN {X 0,Y 89.122,Z 234.356,A -85,B 0,C 180,E1 -29101.754,E2 -29101.754} C_VEL
LIN {X 0,Y 85.302,Z 226.109,A -85,B 0,C 180,E1 -29106.947,E2 -29106.947} C_VEL
LIN {X 0,Y 82.52,Z 220.758,A -85,B 0,C 180,E1 -29111.508,E2 -29111.508} C_VEL
LIN {X 0,Y 80.663,Z 217.456,A -85,B 0,C 180,E1 -29115.012,E2 -29115.012} C_VEL
LIN {X 0,Y 79.015,Z 214.622,A -85,B 0,C 180,E1 -29118.677,E2 -29118.677} C_VEL
LIN {X 0,Y 77.063,Z 211.148,A -85,B 0,C 180,E1 -29124.415,E2 -29124.415} C_VEL
LIN {X 0,Y 74.93,Z 207.451,A -85,B 0,C 180,E1 -29135.64,E2 -29135.64} C_VEL
LIN {X 0,Y 74.877,Z 206.538,A -85,B 0,C 180,E1 -29137.95,E2 -29137.95} C_VEL
LIN {X 0,Y 75.165,Z 206.607,A -85,B 0,C 180,E1 -29147.374,E2 -29147.374} C_VEL
LIN {X 0,Y 77.525,Z 210.882,A -85,B 0,C 180,E1 -29158.828,E2 -29158.828} C_VEL
LIN {X 0,Y 79.759,Z 215.319,A -85,B 0,C 180,E1 -29164.938,E2 -29164.938} C_VEL
LIN {X 0,Y 82.669,Z 220.752,A -85,B 0,C 180,E1 -29170.793,E2 -29170.793} C_VEL
LIN {X 0,Y 86.282,Z 228.298,A -85,B 0,C 180,E1 -29176.565,E2 -29176.565} C_VEL
LIN {X 0,Y 88.138,Z 232.98,A -85,B 0,C 180,E1 -29179.177,E2 -29179.177} C_VEL
LIN {X 0,Y 91.178,Z 245.2,A -85,B 0,C 180,E1 -29183.722,E2 -29183.722} C_VEL
LIN {X 0,Y 91.543,Z 247.693,A -85,B 0,C 180,E1 -29184.368,E2 -29184.368} C_VEL
LIN {X 0,Y 89.414,Z 267.517,A -85,B 0,C 180,E1 -29185.642,E2 -29185.642} C_VEL
LIN {X 0,Y 87.301,Z 281.774,A -85,B 0,C 180,E1 -29186.624,E2 -29186.624} C_VEL
LIN {X 0,Y 84.527,Z 293.552,A -85,B 0,C 180,E1 -29187.944,E2 -29187.944} C_VEL
LIN {X 0,Y 80.974,Z 304.804,A -85,B 0,C 180,E1 -29189.781,E2 -29189.781} C_VEL
LIN {X 0,Y 76.138,Z 316.885,A -85,B 0,C 180,E1 -29192.617,E2 -29192.617} C_VEL
LIN {X 0,Y 70.887,Z 327.804,A -85,B 0,C 180,E1 -29196.337,E2 -29196.337} C_VEL
LIN {X 0,Y 65.355,Z 337.661,A -85,B 0,C 180,E1 -29201.171,E2 -29201.171} C_VEL
LIN {X 0,Y 59.891,Z 346.648,A -85,B 0,C 180,E1 -29207.566,E2 -29207.566} C_VEL
LIN {X 0,Y 54.657,Z 355.462,A -85,B 0,C 180,E1 -29216.874,E2 -29216.874} C_VEL
LIN {X 0,Y 50.982,Z 362.435,A -85,B 0,C 180,E1 -29227.722,E2 -29227.722} C_VEL
LIN {X 0,Y 49.221,Z 368.77,A -85,B 0,C 180,E1 -29241.791,E2 -29241.791} C_VEL
LIN {X 0,Y 49.355,Z 371.633,A -85,B 0,C 180,E1 -29250,E2 -29250} C_VEL
LIN {X 0,Y 49.241,Z 373.791,A -85,B 0,C 180,E1 -29258.205,E2 -29258.205} C_VEL
LIN {X 0,Y 51.32,Z 376.846,A -85,B 0,C 180,E1 -29274.257,E2 -29274.257} C_VEL
LIN {X 0,Y 57.013,Z 378.45,A -85,B 0,C 180,E1 -29288.05,E2 -29288.05} C_VEL
LIN {X 0,Y 65.57,Z 378.604,A -85,B 0,C 180,E1 -29298.614,E2 -29298.614} C_VEL
LIN {X 0,Y 75.878,Z 377.371,A -85,B 0,C 180,E1 -29306.469,E2 -29306.469} C_VEL
LIN {X 0,Y 87.342,Z 374.717,A -85,B 0,C 180,E1 -29312.265,E2 -29312.265} C_VEL
LIN {X 0,Y 99.618,Z 370.495,A -85,B 0,C 180,E1 -29316.51,E2 -29316.51} C_VEL
LIN {X 0,Y 109.175,Z 366.243,A -85,B 0,C 180,E1 -29318.972,E2 -29318.972} C_VEL
LIN {X 0,Y 120.629,Z 359.902,A -85,B 0,C 180,E1 -29321.215,E2 -29321.215} C_VEL
LIN {X 0,Y 127.237,Z 355.551,A -85,B 0,C 180,E1 -29322.332,E2 -29322.332} C_VEL
LIN {X 0,Y 128.41,Z 354.619,A -85,B 0,C 180,E1 -29323.305,E2 -29323.305} C_VEL
LIN {X 0,Y 118.039,Z 361.07,A -85,B 0,C 180,E1 -29325.355,E2 -29325.355} C_VEL
LIN {X 0,Y 116.286,Z 362.007,A -85,B 0,C 180,E1 -29325.741,E2 -29325.741} C_VEL
LIN {X 0,Y 111.205,Z 364.598,A -85,B 0,C 180,E1 -29326.562,E2 -29326.562} C_VEL
LIN {X 0,Y 98.445,Z 369.859,A -85,B 0,C 180,E1 -29327.426,E2 -29327.426} C_VEL
LIN {X 0,Y 91.075,Z 372.148,A -85,B 0,C 180,E1 -29328.385,E2 -29328.385} C_VEL
LIN {X 0,Y 87.576,Z 373.01,A -85,B 0,C 180,E1 -29329.359,E2 -29329.359} C_VEL
LIN {X 0,Y 75.177,Z 375.224,A -85,B 0,C 180,E1 -29334.635,E2 -29334.635} C_VEL
LIN {X 0,Y 63.299,Z 375.863,A -85,B 0,C 180,E1 -29342.227,E2 -29342.227} C_VEL
LIN {X 0,Y 56.824,Z 375.421,A -85,B 0,C 180,E1 -29348.335,E2 -29348.335} C_VEL
LIN {X 0,Y 51.045,Z 374.383,A -85,B 0,C 180,E1 -29355.982,E2 -29355.982} C_VEL
LIN {X 0,Y 45.407,Z 372.197,A -85,B 0,C 180,E1 -29367.665,E2 -29367.665} C_VEL
LIN {X 0,Y 41.998,Z 368.95,A -85,B 0,C 180,E1 -29382.015,E2 -29382.015} C_VEL
LIN {X 0,Y 41.487,Z 363.971,A -85,B 0,C 180,E1 -29399.456,E2 -29399.456} C_VEL
LIN {X 0,Y 43.82,Z 358.201,A -85,B 0,C 180,E1 -29414.209,E2 -29414.209} C_VEL
LIN {X 0,Y 47.535,Z 351.91,A -85,B 0,C 180,E1 -29425.611,E2 -29425.611} C_VEL
LIN {X 0,Y 51.865,Z 345.457,A -85,B 0,C 180,E1 -29433.885,E2 -29433.885} C_VEL
LIN {X 0,Y 57.333,Z 337.214,A -85,B 0,C 180,E1 -29441.293,E2 -29441.293} C_VEL
LIN {X 0,Y 63.792,Z 326.724,A -85,B 0,C 180,E1 -29447.636,E2 -29447.636} C_VEL
LIN {X 0,Y 69.474,Z 316.022,A -85,B 0,C 180,E1 -29451.991,E2 -29451.991} C_VEL
LIN {X 0,Y 74.442,Z 304.911,A -85,B 0,C 180,E1 -29455.141,E2 -29455.141} C_VEL
LIN {X 0,Y 78.867,Z 292.699,A -85,B 0,C 180,E1 -29457.543,E2 -29457.543} C_VEL
LIN {X 0,Y 82.368,Z 279.309,A -85,B 0,C 180,E1 -29459.371,E2 -29459.371} C_VEL
LIN {X 0,Y 84.83,Z 265.324,A -85,B 0,C 180,E1 -29460.491,E2 -29460.491} C_VEL
LIN {X 0,Y 87.43,Z 244.22,A -85,B 0,C 180,E1 -29461.652,E2 -29461.652} C_VEL
LIN {X 0,Y 85.161,Z 238.182,A -85,B 0,C 180,E1 -29464.851,E2 -29464.851} C_VEL
LIN {X 0,Y 81.806,Z 230.193,A -85,B 0,C 180,E1 -29470.353,E2 -29470.353} C_VEL
LIN {X 0,Y 78.698,Z 223.985,A -85,B 0,C 180,E1 -29476.529,E2 -29476.529} C_VEL
LIN {X 0,Y 77.046,Z 220.891,A -85,B 0,C 180,E1 -29480.722,E2 -29480.722} C_VEL
LIN {X 0,Y 75.489,Z 217.811,A -85,B 0,C 180,E1 -29486.043,E2 -29486.043} C_VEL
LIN {X 0,Y 73.801,Z 214.194,A -85,B 0,C 180,E1 -29497.103,E2 -29497.103} C_VEL
LIN {X 0,Y 73.806,Z 213.524,A -85,B 0,C 180,E1 -29498.866,E2 -29498.866} C_VEL
LIN {X 0,Y 74.014,Z 213.582,A -85,B 0,C 180,E1 -29506.418,E2 -29506.418} C_VEL
LIN {X 0,Y 75.872,Z 217.413,A -85,B 0,C 180,E1 -29517.045,E2 -29517.045} C_VEL
LIN {X 0,Y 77.764,Z 221.69,A -85,B 0,C 180,E1 -29523.108,E2 -29523.108} C_VEL
LIN {X 0,Y 80.208,Z 226.721,A -85,B 0,C 180,E1 -29528.652,E2 -29528.652} C_VEL
LIN {X 0,Y 83.212,Z 233.709,A -85,B 0,C 180,E1 -29534.224,E2 -29534.224} C_VEL
LIN {X 0,Y 84.554,Z 237.616,A -85,B 0,C 180,E1 -29536.467,E2 -29536.467} C_VEL
LIN {X 0,Y 87.013,Z 248.694,A -85,B 0,C 180,E1 -29540.762,E2 -29540.762} C_VEL
LIN {X 0,Y 87.119,Z 249.285,A -85,B 0,C 180,E1 -29540.956,E2 -29540.956} C_VEL
LIN {X 0,Y 83.52,Z 277.461,A -85,B 0,C 180,E1 -29542.632,E2 -29542.632} C_VEL
LIN {X 0,Y 80.693,Z 290.308,A -85,B 0,C 180,E1 -29543.865,E2 -29543.865} C_VEL
LIN {X 0,Y 76.969,Z 302.363,A -85,B 0,C 180,E1 -29545.62,E2 -29545.62} C_VEL
LIN {X 0,Y 71.845,Z 314.85,A -85,B 0,C 180,E1 -29548.31,E2 -29548.31} C_VEL
LIN {X 0,Y 66.248,Z 326.051,A -85,B 0,C 180,E1 -29551.931,E2 -29551.931} C_VEL
LIN {X 0,Y 60.277,Z 336.183,A -85,B 0,C 180,E1 -29556.717,E2 -29556.717} C_VEL
LIN {X 0,Y 54.888,Z 344.531,A -85,B 0,C 180,E1 -29562.588,E2 -29562.588} C_VEL
LIN {X 0,Y 48.854,Z 353.603,A -85,B 0,C 180,E1 -29572.31,E2 -29572.31} C_VEL
LIN {X 0,Y 44.491,Z 360.879,A -85,B 0,C 180,E1 -29584.252,E2 -29584.252} C_VEL
LIN {X 0,Y 42.5,Z 365.773,A -85,B 0,C 180,E1 -29595.638,E2 -29595.638} C_VEL
LIN {X 0,Y 42.298,Z 370.473,A -85,B 0,C 180,E1 -29610,E2 -29610} C_VEL
LIN {X 0,Y 42.286,Z 372.796,A -85,B 0,C 180,E1 -29619.567,E2 -29619.567} C_VEL
LIN {X 0,Y 44.951,Z 376.053,A -85,B 0,C 180,E1 -29637.971,E2 -29637.971} C_VEL
LIN {X 0,Y 51.604,Z 377.831,A -85,B 0,C 180,E1 -29652.918,E2 -29652.918} C_VEL
LIN {X 0,Y 61.1,Z 378.249,A -85,B 0,C 180,E1 -29663.626,E2 -29663.626} C_VEL
LIN {X 0,Y 72.197,Z 377.219,A -85,B 0,C 180,E1 -29671.174,E2 -29671.174} C_VEL
LIN {X 0,Y 84.267,Z 374.795,A -85,B 0,C 180,E1 -29676.551,E2 -29676.551} C_VEL
LIN {X 0,Y 97.017,Z 370.886,A -85,B 0,C 180,E1 -29680.342,E2 -29680.342} C_VEL
LIN {X 0,Y 106.541,Z 366.982,A -85,B 0,C 180,E1 -29682.449,E2 -29682.449} C_VEL
LIN {X 0,Y 110.093,Z 365.271,A -85,B 0,C 180,E1 -29683.244,E2 -29683.244} C_VEL
LIN {X 0,Y 97.826,Z 370.126,A -85,B 0,C 180,E1 -29686.151,E2 -29686.151} C_VEL
LIN {X 0,Y 87.576,Z 373.01,A -85,B 0,C 180,E1 -29689.359,E2 -29689.359} C_VEL
LIN {X 0,Y 82.237,Z 374.187,A -85,B 0,C 180,E1 -29690.877,E2 -29690.877} C_VEL
LIN {X 0,Y 72.721,Z 375.614,A -85,B 0,C 180,E1 -29692.627,E2 -29692.627} C_VEL
LIN {X 0,Y 63.235,Z 376.27,A -85,B 0,C 180,E1 -29694.931,E2 -29694.931} C_VEL
LIN {X 0,Y 58.08,Z 376.143,A -85,B 0,C 180,E1 -29697.627,E2 -29697.627} C_VEL
LIN {X 0,Y 49.431,Z 375.267,A -85,B 0,C 180,E1 -29705.602,E2 -29705.602} C_VEL
LIN {X 0,Y 43.455,Z 373.863,A -85,B 0,C 180,E1 -29713.983,E2 -29713.983} C_VEL
LIN {X 0,Y 36.87,Z 370.592,A -85,B 0,C 180,E1 -29730.614,E2 -29730.614} C_VEL
LIN {X 0,Y 34.217,Z 365.776,A -85,B 0,C 180,E1 -29751.963,E2 -29751.963} C_VEL
LIN {X 0,Y 35.731,Z 360.199,A -85,B 0,C 180,E1 -29770.994,E2 -29770.994} C_VEL
LIN {X 0,Y 39.385,Z 354.316,A -85,B 0,C 180,E1 -29784.882,E2 -29784.882} C_VEL
LIN {X 0,Y 44.914,Z 346.693,A -85,B 0,C 180,E1 -29796.74,E2 -29796.74} C_VEL
LIN {X 0,Y 51.626,Z 337.357,A -85,B 0,C 180,E1 -29805.799,E2 -29805.799} C_VEL
LIN {X 0,Y 57.676,Z 328.292,A -85,B 0,C 180,E1 -29811.442,E2 -29811.442} C_VEL
LIN {X 0,Y 64.012,Z 317.33,A -85,B 0,C 180,E1 -29816.051,E2 -29816.051} C_VEL
LIN {X 0,Y 69.791,Z 305.2,A -85,B 0,C 180,E1 -29819.401,E2 -29819.401} C_VEL
LIN {X 0,Y 74.274,Z 293.434,A -85,B 0,C 180,E1 -29821.616,E2 -29821.616} C_VEL
LIN {X 0,Y 77.873,Z 280.742,A -85,B 0,C 180,E1 -29823.273,E2 -29823.273} C_VEL
LIN {X 0,Y 80.494,Z 266.802,A -85,B 0,C 180,E1 -29824.388,E2 -29824.388} C_VEL
LIN {X 0,Y 83.147,Z 246.766,A -85,B 0,C 180,E1 -29825.38,E2 -29825.38} C_VEL
LIN {X 0,Y 80.245,Z 238.716,A -85,B 0,C 180,E1 -29830.545,E2 -29830.545} C_VEL
LIN {X 0,Y 77.983,Z 233.254,A -85,B 0,C 180,E1 -29835.215,E2 -29835.215} C_VEL
LIN {X 0,Y 76.112,Z 229.161,A -85,B 0,C 180,E1 -29839.94,E2 -29839.94} C_VEL
LIN {X 0,Y 74.883,Z 226.557,A -85,B 0,C 180,E1 -29843.919,E2 -29843.919} C_VEL
LIN {X 0,Y 73.911,Z 224.418,A -85,B 0,C 180,E1 -29847.895,E2 -29847.895} C_VEL
LIN {X 0,Y 72.741,Z 220.553,A -85,B 0,C 180,E1 -29859.838,E2 -29859.838} C_VEL
LIN {X 0,Y 72.901,Z 220.668,A -85,B 0,C 180,E1 -29865.822,E2 -29865.822} C_VEL
LIN {X 0,Y 74.272,Z 223.898,A -85,B 0,C 180,E1 -29875.079,E2 -29875.079} C_VEL
LIN {X 0,Y 75.762,Z 227.859,A -85,B 0,C 180,E1 -29880.907,E2 -29880.907} C_VEL
LIN {X 0,Y 77.649,Z 232.2,A -85,B 0,C 180,E1 -29885.967,E2 -29885.967} C_VEL
LIN {X 0,Y 80.164,Z 238.776,A -85,B 0,C 180,E1 -29891.459,E2 -29891.459} C_VEL
LIN {X 0,Y 81.126,Z 242.133,A -85,B 0,C 180,E1 -29893.442,E2 -29893.442} C_VEL
LIN {X 0,Y 82.835,Z 251.032,A -85,B 0,C 180,E1 -29897.146,E2 -29897.146} C_VEL
LIN {X 0,Y 79.251,Z 277.461,A -85,B 0,C 180,E1 -29898.637,E2 -29898.637} C_VEL
LIN {X 0,Y 76.178,Z 290.641,A -85,B 0,C 180,E1 -29899.841,E2 -29899.841} C_VEL
LIN {X 0,Y 72.24,Z 302.617,A -85,B 0,C 180,E1 -29901.519,E2 -29901.519} C_VEL
LIN {X 0,Y 66.508,Z 315.719,A -85,B 0,C 180,E1 -29904.298,E2 -29904.298} C_VEL
LIN {X 0,Y 60.722,Z 326.479,A -85,B 0,C 180,E1 -29907.766,E2 -29907.766} C_VEL
LIN {X 0,Y 54.297,Z 336.596,A -85,B 0,C 180,E1 -29912.718,E2 -29912.718} C_VEL
LIN {X 0,Y 47.878,Z 345.6,A -85,B 0,C 180,E1 -29919.588,E2 -29919.588} C_VEL
LIN {X 0,Y 41.502,Z 354.433,A -85,B 0,C 180,E1 -29930.578,E2 -29930.578} C_VEL
LIN {X 0,Y 37.012,Z 361.448,A -85,B 0,C 180,E1 -29944.707,E2 -29944.707} C_VEL
LIN {X 0,Y 35.094,Z 367.803,A -85,B 0,C 180,E1 -29964.259,E2 -29964.259} C_VEL
LIN {X 0,Y 35.25,Z 369.303,A -85,B 0,C 180,E1 -29969.999,E2 -29969.999} C_VEL
LIN {X 0,Y 35.317,Z 370.624,A -85,B 0,C 180,E1 -29975.715,E2 -29975.715} C_VEL
LIN {X 0,Y 36.444,Z 373.655,A -85,B 0,C 180,E1 -29992.685,E2 -29992.685} C_VEL
LIN {X 0,Y 42.312,Z 376.39,A -85,B 0,C 180,E1 -30011.636,E2 -30011.636} C_VEL
LIN {X 0,Y 51.721,Z 377.685,A -85,B 0,C 180,E1 -30024.615,E2 -30024.615} C_VEL
LIN {X 0,Y 62.969,Z 377.603,A -85,B 0,C 180,E1 -30033.236,E2 -30033.236} C_VEL
LIN {X 0,Y 75.298,Z 376.147,A -85,B 0,C 180,E1 -30038.962,E2 -30038.962} C_VEL
LIN {X 0,Y 88.242,Z 373.214,A -85,B 0,C 180,E1 -30042.886,E2 -30042.886} C_VEL
LIN {X 0,Y 87.637,Z 373.27,A -85,B 0,C 180,E1 -30044.222,E2 -30044.222} C_VEL
LIN {X 0,Y 79.399,Z 374.899,A -85,B 0,C 180,E1 -30046.82,E2 -30046.82} C_VEL
LIN {X 0,Y 71.369,Z 375.902,A -85,B 0,C 180,E1 -30049.975,E2 -30049.975} C_VEL
LIN {X 0,Y 63.601,Z 376.29,A -85,B 0,C 180,E1 -30053.99,E2 -30053.99} C_VEL
LIN {X 0,Y 58.08,Z 376.143,A -85,B 0,C 180,E1 -30057.627,E2 -30057.627} C_VEL
LIN {X 0,Y 53.075,Z 375.874,A -85,B 0,C 180,E1 -30060.84,E2 -30060.84} C_VEL
LIN {X 0,Y 44.176,Z 374.761,A -85,B 0,C 180,E1 -30065.819,E2 -30065.819} C_VEL
LIN {X 0,Y 37.35,Z 373.303,A -85,B 0,C 180,E1 -30071.195,E2 -30071.195} C_VEL
LIN {X 0,Y 33.106,Z 371.873,A -85,B 0,C 180,E1 -30077.509,E2 -30077.509} C_VEL
LIN {X 0,Y 32.009,Z 371.316,A -85,B 0,C 180,E1 -30080.239,E2 -30080.239} C_VEL
LIN {X 0,Y 27.752,Z 367.523,A -85,B 0,C 180,E1 -30100.561,E2 -30100.561} C_VEL
LIN {X 0,Y 27.519,Z 362.66,A -85,B 0,C 180,E1 -30123.458,E2 -30123.458} C_VEL
LIN {X 0,Y 30.992,Z 356.645,A -85,B 0,C 180,E1 -30143.49,E2 -30143.49} C_VEL
LIN {X 0,Y 36.623,Z 349.451,A -85,B 0,C 180,E1 -30158.239,E2 -30158.239} C_VEL
LIN {X 0,Y 43.811,Z 340.659,A -85,B 0,C 180,E1 -30168.713,E2 -30168.713} C_VEL
LIN {X 0,Y 51.006,Z 331.035,A -85,B 0,C 180,E1 -30175.506,E2 -30175.506} C_VEL
LIN {X 0,Y 57.705,Z 320.576,A -85,B 0,C 180,E1 -30180.158,E2 -30180.158} C_VEL
LIN {X 0,Y 63.795,Z 309.279,A -85,B 0,C 180,E1 -30183.424,E2 -30183.424} C_VEL
LIN {X 0,Y 68.913,Z 297.515,A -85,B 0,C 180,E1 -30185.68,E2 -30185.68} C_VEL
LIN {X 0,Y 73.169,Z 284.193,A -85,B 0,C 180,E1 -30187.477,E2 -30187.477} C_VEL
LIN {X 0,Y 76.084,Z 271.234,A -85,B 0,C 180,E1 -30188.563,E2 -30188.563} C_VEL
LIN {X 0,Y 79.123,Z 249.11,A -85,B 0,C 180,E1 -30189.708,E2 -30189.708} C_VEL
LIN {X 0,Y 76.569,Z 241.532,A -85,B 0,C 180,E1 -30195.34,E2 -30195.34} C_VEL
LIN {X 0,Y 74.591,Z 236.294,A -85,B 0,C 180,E1 -30200.85,E2 -30200.85} C_VEL
LIN {X 0,Y 73.286,Z 233.127,A -85,B 0,C 180,E1 -30205.642,E2 -30205.642} C_VEL
LIN {X 0,Y 72.509,Z 231.125,A -85,B 0,C 180,E1 -30209.36,E2 -30209.36} C_VEL
LIN {X 0,Y 71.679,Z 227.554,A -85,B 0,C 180,E1 -30220.834,E2 -30220.834} C_VEL
LIN {X 0,Y 71.815,Z 227.844,A -85,B 0,C 180,E1 -30225.587,E2 -30225.587} C_VEL
LIN {X 0,Y 72.795,Z 230.592,A -85,B 0,C 180,E1 -30233.418,E2 -30233.418} C_VEL
LIN {X 0,Y 74.005,Z 234.42,A -85,B 0,C 180,E1 -30239.098,E2 -30239.098} C_VEL
LIN {X 0,Y 75.332,Z 238.088,A -85,B 0,C 180,E1 -30243.42,E2 -30243.42} C_VEL
LIN {X 0,Y 77.358,Z 244.002,A -85,B 0,C 180,E1 -30248.594,E2 -30248.594} C_VEL
LIN {X 0,Y 77.978,Z 246.851,A -85,B 0,C 180,E1 -30250.262,E2 -30250.262} C_VEL
LIN {X 0,Y 78.906,Z 252.797,A -85,B 0,C 180,E1 -30252.922,E2 -30252.922} C_VEL
LIN {X 0,Y 75.476,Z 277.073,A -85,B 0,C 180,E1 -30254.202,E2 -30254.202} C_VEL
LIN {X 0,Y 72.391,Z 289.905,A -85,B 0,C 180,E1 -30255.254,E2 -30255.254} C_VEL
LIN {X 0,Y 67.929,Z 302.816,A -85,B 0,C 180,E1 -30256.862,E2 -30256.862} C_VEL
LIN {X 0,Y 62.337,Z 315.029,A -85,B 0,C 180,E1 -30259.229,E2 -30259.229} C_VEL
LIN {X 0,Y 55.881,Z 326.422,A -85,B 0,C 180,E1 -30262.643,E2 -30262.643} C_VEL
LIN {X 0,Y 49.355,Z 336.016,A -85,B 0,C 180,E1 -30267.128,E2 -30267.128} C_VEL
LIN {X 0,Y 42.357,Z 345.045,A -85,B 0,C 180,E1 -30273.94,E2 -30273.94} C_VEL
LIN {X 0,Y 35.209,Z 353.881,A -85,B 0,C 180,E1 -30285.682,E2 -30285.682} C_VEL
LIN {X 0,Y 30.082,Z 360.916,A -85,B 0,C 180,E1 -30302.143,E2 -30302.143} C_VEL
LIN {X 0,Y 28.05,Z 366.478,A -85,B 0,C 180,E1 -30322.81,E2 -30322.81} C_VEL
LIN {X 0,Y 28.202,Z 368.06,A -85,B 0,C 180,E1 -30329.999,E2 -30329.999} C_VEL
LIN {X 0,Y 28.35,Z 369.459,A -85,B 0,C 180,E1 -30337.413,E2 -30337.413} C_VEL
LIN {X 0,Y 30.056,Z 372.64,A -85,B 0,C 180,E1 -30357.882,E2 -30357.882} C_VEL
LIN {X 0,Y 37.305,Z 375.598,A -85,B 0,C 180,E1 -30378.899,E2 -30378.899} C_VEL
LIN {X 0,Y 47.96,Z 377.143,A -85,B 0,C 180,E1 -30391.547,E2 -30391.547} C_VEL
LIN {X 0,Y 60.096,Z 377.263,A -85,B 0,C 180,E1 -30399.32,E2 -30399.32} C_VEL
LIN {X 0,Y 67.863,Z 376.69,A -85,B 0,C 180,E1 -30402.463,E2 -30402.463} C_VEL
LIN {X 0,Y 70.314,Z 376.361,A -85,B 0,C 180,E1 -30404.054,E2 -30404.054} C_VEL
LIN {X 0,Y 57.116,Z 376.659,A -85,B 0,C 180,E1 -30409.857,E2 -30409.857} C_VEL
LIN {X 0,Y 49.387,Z 376.067,A -85,B 0,C 180,E1 -30414.954,E2 -30414.954} C_VEL
LIN {X 0,Y 42.19,Z 374.854,A -85,B 0,C 180,E1 -30421.871,E2 -30421.871} C_VEL
LIN {X 0,Y 33.114,Z 371.905,A -85,B 0,C 180,E1 -30437.244,E2 -30437.244} C_VEL
LIN {X 0,Y 32.009,Z 371.316,A -85,B 0,C 180,E1 -30440.239,E2 -30440.239} C_VEL
LIN {X 0,Y 28.857,Z 369.583,A -85,B 0,C 180,E1 -30449.021,E2 -30449.021} C_VEL
LIN {X 0,Y 23.786,Z 366.027,A -85,B 0,C 180,E1 -30465.999,E2 -30465.999} C_VEL
LIN {X 0,Y 21.511,Z 362.64,A -85,B 0,C 180,E1 -30483.518,E2 -30483.518} C_VEL
LIN {X 0,Y 21.937,Z 359.789,A -85,B 0,C 180,E1 -30497.356,E2 -30497.356} C_VEL
LIN {X 0,Y 22.57,Z 358.777,A -85,B 0,C 180,E1 -30501.496,E2 -30501.496} C_VEL
LIN {X 0,Y 28.635,Z 351.878,A -85,B 0,C 180,E1 -30520.98,E2 -30520.98} C_VEL
LIN {X 0,Y 36.159,Z 343.736,A -85,B 0,C 180,E1 -30532.876,E2 -30532.876} C_VEL
LIN {X 0,Y 44.689,Z 333.518,A -85,B 0,C 180,E1 -30540.738,E2 -30540.738} C_VEL
LIN {X 0,Y 52.016,Z 323.263,A -85,B 0,C 180,E1 -30545.298,E2 -30545.298} C_VEL
LIN {X 0,Y 58.213,Z 312.844,A -85,B 0,C 180,E1 -30548.224,E2 -30548.224} C_VEL
LIN {X 0,Y 64.205,Z 300.284,A -85,B 0,C 180,E1 -30550.536,E2 -30550.536} C_VEL
LIN {X 0,Y 68.672,Z 288.029,A -85,B 0,C 180,E1 -30552.078,E2 -30552.078} C_VEL
LIN {X 0,Y 71.976,Z 275.273,A -85,B 0,C 180,E1 -30553.118,E2 -30553.118} C_VEL
LIN {X 0,Y 74.975,Z 256.244,A -85,B 0,C 180,E1 -30554.016,E2 -30554.016} C_VEL
LIN {X 0,Y 75.512,Z 251.825,A -85,B 0,C 180,E1 -30554.317,E2 -30554.317} C_VEL
LIN {X 0,Y 73.677,Z 245.51,A -85,B 0,C 180,E1 -30559.662,E2 -30559.662} C_VEL
LIN {X 0,Y 72.335,Z 241.363,A -85,B 0,C 180,E1 -30564.735,E2 -30564.735} C_VEL
LIN {X 0,Y 71.175,Z 237.877,A -85,B 0,C 180,E1 -30570.764,E2 -30570.764} C_VEL
LIN {X 0,Y 70.642,Z 234.54,A -85,B 0,C 180,E1 -30581.592,E2 -30581.592} C_VEL
LIN {X 0,Y 70.708,Z 234.823,A -85,B 0,C 180,E1 -30584.674,E2 -30584.674} C_VEL
LIN {X 0,Y 71.326,Z 237.058,A -85,B 0,C 180,E1 -30591.37,E2 -30591.37} C_VEL
LIN {X 0,Y 72.234,Z 240.618,A -85,B 0,C 180,E1 -30596.744,E2 -30596.744} C_VEL
LIN {X 0,Y 73.178,Z 243.904,A -85,B 0,C 180,E1 -30600.705,E2 -30600.705} C_VEL
LIN {X 0,Y 74.629,Z 249.008,A -85,B 0,C 180,E1 -30605.405,E2 -30605.405} C_VEL
LIN {X 0,Y 75.424,Z 254.516,A -85,B 0,C 180,E1 -30608.275,E2 -30608.275} C_VEL
LIN {X 0,Y 72.117,Z 276.94,A -85,B 0,C 180,E1 -30609.349,E2 -30609.349} C_VEL
LIN {X 0,Y 68.749,Z 290.28,A -85,B 0,C 180,E1 -30610.284,E2 -30610.284} C_VEL
LIN {X 0,Y 64.552,Z 301.963,A -85,B 0,C 180,E1 -30611.52,E2 -30611.52} C_VEL
LIN {X 0,Y 58.726,Z 314.238,A -85,B 0,C 180,E1 -30613.506,E2 -30613.506} C_VEL
LIN {X 0,Y 52.534,Z 324.713,A -85,B 0,C 180,E1 -30616.111,E2 -30616.111} C_VEL
LIN {X 0,Y 44.99,Z 335.323,A -85,B 0,C 180,E1 -30620.4,E2 -30620.4} C_VEL
LIN {X 0,Y 37.377,Z 344.371,A -85,B 0,C 180,E1 -30626.729,E2 -30626.729} C_VEL
LIN {X 0,Y 29.294,Z 353.247,A -85,B 0,C 180,E1 -30638.765,E2 -30638.765} C_VEL
LIN {X 0,Y 23.256,Z 360.336,A -85,B 0,C 180,E1 -30658.071,E2 -30658.071} C_VEL
LIN {X 0,Y 21.125,Z 366.72,A -85,B 0,C 180,E1 -30689.999,E2 -30689.999} C_VEL
LIN {X 0,Y 21.43,Z 368.301,A -85,B 0,C 180,E1 -30700.28,E2 -30700.28} C_VEL
LIN {X 0,Y 24.046,Z 371.616,A -85,B 0,C 180,E1 -30725.769,E2 -30725.769} C_VEL
LIN {X 0,Y 33.09,Z 374.756,A -85,B 0,C 180,E1 -30748.162,E2 -30748.162} C_VEL
LIN {X 0,Y 45.014,Z 376.516,A -85,B 0,C 180,E1 -30759.516,E2 -30759.516} C_VEL
LIN {X 0,Y 51.403,Z 376.881,A -85,B 0,C 180,E1 -30763.145,E2 -30763.145} C_VEL
LIN {X 0,Y 51.859,Z 376.852,A -85,B 0,C 180,E1 -30764.272,E2 -30764.272} C_VEL
LIN {X 0,Y 41.882,Z 375.633,A -85,B 0,C 180,E1 -30770.338,E2 -30770.338} C_VEL
LIN {X 0,Y 32.552,Z 373.456,A -85,B 0,C 180,E1 -30779.997,E2 -30779.997} C_VEL
LIN {X 0,Y 24.738,Z 370.266,A -85,B 0,C 180,E1 -30796.501,E2 -30796.501} C_VEL
LIN {X 0,Y 20.225,Z 365.569,A -85,B 0,C 180,E1 -30825.977,E2 -30825.977} C_VEL
LIN {X 0,Y 21.7,Z 360.045,A -85,B 0,C 180,E1 -30856.297,E2 -30856.297} C_VEL
LIN {X 0,Y 22.57,Z 358.777,A -85,B 0,C 180,E1 -30861.496,E2 -30861.496} C_VEL
LIN {X 0,Y 23.937,Z 356.726,A -85,B 0,C 180,E1 -30869.076,E2 -30869.076} C_VEL
LIN {X 0,Y 25.757,Z 353.438,A -85,B 0,C 180,E1 -30879.699,E2 -30879.699} C_VEL
LIN {X 0,Y 31.107,Z 344.943,A -85,B 0,C 180,E1 -30899.503,E2 -30899.503} C_VEL
LIN {X 0,Y 34.434,Z 340.909,A -85,B 0,C 180,E1 -30904.488,E2 -30904.488} C_VEL
LIN {X 0,Y 35.693,Z 339.497,A -85,B 0,C 180,E1 -30905.536,E2 -30905.536} C_VEL
LIN {X 0,Y 44.593,Z 328.85,A -85,B 0,C 180,E1 -30910.656,E2 -30910.656} C_VEL
LIN {X 0,Y 52.155,Z 317.784,A -85,B 0,C 180,E1 -30913.678,E2 -30913.678} C_VEL
LIN {X 0,Y 58.846,Z 305.507,A -85,B 0,C 180,E1 -30915.773,E2 -30915.773} C_VEL
LIN {X 0,Y 63.986,Z 293.408,A -85,B 0,C 180,E1 -30917.11,E2 -30917.11} C_VEL
LIN {X 0,Y 68.057,Z 279.977,A -85,B 0,C 180,E1 -30918.19,E2 -30918.19} C_VEL
LIN {X 0,Y 70.736,Z 266.718,A -85,B 0,C 180,E1 -30918.765,E2 -30918.765} C_VEL
LIN {X 0,Y 72.409,Z 254.789,A -85,B 0,C 180,E1 -30919.242,E2 -30919.242} C_VEL
LIN {X 0,Y 71.276,Z 250.047,A -85,B 0,C 180,E1 -30923.93,E2 -30923.93} C_VEL
LIN {X 0,Y 70.274,Z 246.295,A -85,B 0,C 180,E1 -30929.14,E2 -30929.14} C_VEL
LIN {X 0,Y 69.757,Z 244.363,A -85,B 0,C 180,E1 -30933.229,E2 -30933.229} C_VEL
LIN {X 0,Y 69.61,Z 241.561,A -85,B 0,C 180,E1 -30942.37,E2 -30942.37} C_VEL
LIN {X 0,Y 69.945,Z 243.521,A -85,B 0,C 180,E1 -30949.213,E2 -30949.213} C_VEL
LIN {X 0,Y 70.636,Z 247.094,A -85,B 0,C 180,E1 -30954.654,E2 -30954.654} C_VEL
LIN {X 0,Y 71.225,Z 249.834,A -85,B 0,C 180,E1 -30957.97,E2 -30957.97} C_VEL
LIN {X 0,Y 72.178,Z 254.287,A -85,B 0,C 180,E1 -30962.153,E2 -30962.153} C_VEL
LIN {X 0,Y 72.363,Z 256.737,A -85,B 0,C 180,E1 -30963.389,E2 -30963.389} C_VEL
LIN {X 0,Y 69.17,Z 277.049,A -85,B 0,C 180,E1 -30964.11,E2 -30964.11} C_VEL
LIN {X 0,Y 65.756,Z 290.102,A -85,B 0,C 180,E1 -30964.817,E2 -30964.817} C_VEL
LIN {X 0,Y 60.933,Z 302.845,A -85,B 0,C 180,E1 -30965.845,E2 -30965.845} C_VEL
LIN {X 0,Y 54.844,Z 314.995,A -85,B 0,C 180,E1 -30967.364,E2 -30967.364} C_VEL
LIN {X 0,Y 48.1,Z 325.73,A -85,B 0,C 180,E1 -30969.508,E2 -30969.508} C_VEL
LIN {X 0,Y 39.714,Z 336.539,A -85,B 0,C 180,E1 -30973.268,E2 -30973.268} C_VEL
LIN {X 0,Y 31.567,Z 345.313,A -85,B 0,C 180,E1 -30978.877,E2 -30978.877} C_VEL
LIN {X 0,Y 24.014,Z 352.614,A -85,B 0,C 180,E1 -30988.599,E2 -30988.599} C_VEL
LIN {X 0,Y 16.652,Z 359.753,A -85,B 0,C 180,E1 -31010.722,E2 -31010.722} C_VEL
LIN {X 0,Y 14.058,Z 365.371,A -85,B 0,C 180,E1 -31049.999,E2 -31049.999} C_VEL
LIN {X 0,Y 14.631,Z 367.104,A -85,B 0,C 180,E1 -31066.09,E2 -31066.09} C_VEL
LIN {X 0,Y 18.789,Z 370.457,A -85,B 0,C 180,E1 -31098.426,E2 -31098.426} C_VEL
LIN {X 0,Y 29.969,Z 373.893,A -85,B 0,C 180,E1 -31119.721,E2 -31119.721} C_VEL
LIN {X 0,Y 33.238,Z 374.436,A -85,B 0,C 180,E1 -31124.811,E2 -31124.811} C_VEL
LIN {X 0,Y 21.084,Z 370.62,A -85,B 0,C 180,E1 -31140.237,E2 -31140.237} C_VEL
LIN {X 0,Y 14.092,Z 366.329,A -85,B 0,C 180,E1 -31169.908,E2 -31169.908} C_VEL
LIN {X 0,Y 14.337,Z 360.536,A -85,B 0,C 180,E1 -31218.616,E2 -31218.616} C_VEL
LIN {X 0,Y 21.934,Z 352.996,A -85,B 0,C 180,E1 -31248.688,E2 -31248.688} C_VEL
LIN {X 0,Y 30.217,Z 345.199,A -85,B 0,C 180,E1 -31260.782,E2 -31260.782} C_VEL
LIN {X 0,Y 35.693,Z 339.497,A -85,B 0,C 180,E1 -31265.536,E2 -31265.536} C_VEL
LIN {X 0,Y 39.141,Z 335.281,A -85,B 0,C 180,E1 -31268.748,E2 -31268.748} C_VEL
LIN {X 0,Y 43.85,Z 327.922,A -85,B 0,C 180,E1 -31275.02,E2 -31275.02} C_VEL
LIN {X 0,Y 48.41,Z 319.977,A -85,B 0,C 180,E1 -31280.073,E2 -31280.073} C_VEL
LIN {X 0,Y 51.39,Z 314.882,A -85,B 0,C 180,E1 -31281.528,E2 -31281.528} C_VEL
LIN {X 0,Y 57.343,Z 303.726,A -85,B 0,C 180,E1 -31282.588,E2 -31282.588} C_VEL
LIN {X 0,Y 62.273,Z 291.787,A -85,B 0,C 180,E1 -31283.35,E2 -31283.35} C_VEL
LIN {X 0,Y 66.377,Z 277.952,A -85,B 0,C 180,E1 -31284.055,E2 -31284.055} C_VEL
LIN {X 0,Y 69.137,Z 262.847,A -85,B 0,C 180,E1 -31284.412,E2 -31284.412} C_VEL
LIN {X 0,Y 69.832,Z 257.9,A -85,B 0,C 180,E1 -31284.608,E2 -31284.608} C_VEL
LIN {X 0,Y 68.985,Z 253.533,A -85,B 0,C 180,E1 -31289.986,E2 -31289.986} C_VEL
LIN {X 0,Y 68.579,Z 251.242,A -85,B 0,C 180,E1 -31294.315,E2 -31294.315} C_VEL
LIN {X 0,Y 68.509,Z 248.956,A -85,B 0,C 180,E1 -31302.077,E2 -31302.077} C_VEL
LIN {X 0,Y 68.594,Z 249.543,A -85,B 0,C 180,E1 -31305.597,E2 -31305.597} C_VEL
LIN {X 0,Y 68.749,Z 251.036,A -85,B 0,C 180,E1 -31308.764,E2 -31308.764} C_VEL
LIN {X 0,Y 69.348,Z 255.062,A -85,B 0,C 180,E1 -31314.386,E2 -31314.386} C_VEL
LIN {X 0,Y 69.869,Z 258.554,A -85,B 0,C 180,E1 -31317.924,E2 -31317.924} C_VEL
LIN {X 0,Y 67.014,Z 276.41,A -85,B 0,C 180,E1 -31318.445,E2 -31318.445} C_VEL
LIN {X 0,Y 63.833,Z 288.567,A -85,B 0,C 180,E1 -31318.839,E2 -31318.839} C_VEL
LIN {X 0,Y 59.302,Z 300.808,A -85,B 0,C 180,E1 -31319.352,E2 -31319.352} C_VEL
LIN {X 0,Y 52.904,Z 313.6,A -85,B 0,C 180,E1 -31320.191,E2 -31320.191} C_VEL
LIN {X 0,Y 45.696,Z 324.906,A -85,B 0,C 180,E1 -31321.413,E2 -31321.413} C_VEL
LIN {X 0,Y 38.708,Z 333.807,A -85,B 0,C 180,E1 -31323.013,E2 -31323.013} C_VEL
LIN {X 0,Y 30.035,Z 342.973,A -85,B 0,C 180,E1 -31326.021,E2 -31326.021} C_VEL
LIN {X 0,Y 19.882,Z 351.918,A -85,B 0,C 180,E1 -31333.57,E2 -31333.57} C_VEL
LIN {X 0,Y 10.665,Z 359.084,A -85,B 0,C 180,E1 -31354.539,E2 -31354.539} C_VEL
LIN {X 0,Y 7.035,Z 364.008,A -85,B 0,C 180,E1 -31412.17,E2 -31412.17} C_VEL
LIN {X 0,Y 8.328,Z 365.888,A -85,B 0,C 180,E1 -31442.429,E2 -31442.429} C_VEL
LIN {X 0,Y 15.067,Z 369.295,A -85,B 0,C 180,E1 -31478.891,E2 -31478.891} C_VEL
LIN {X 0,Y 14.465,Z 368.959,A -85,B 0,C 180,E1 -31486.341,E2 -31486.341} C_VEL
LIN {X 0,Y 6.306,Z 364.131,A -85,B 0,C 180,E1 -31533.292,E2 -31533.292} C_VEL
LIN {X 0,Y 10.501,Z 358.134,A -85,B 0,C 180,E1 -31609.551,E2 -31609.551} C_VEL
LIN {X 0,Y 18.571,Z 352.043,A -85,B 0,C 180,E1 -31626.403,E2 -31626.403} C_VEL
LIN {X 0,Y 27.835,Z 344.054,A -85,B 0,C 180,E1 -31633.975,E2 -31633.975} C_VEL
LIN {X 0,Y 37.732,Z 333.768,A -85,B 0,C 180,E1 -31638.163,E2 -31638.163} C_VEL
LIN {X 0,Y 45.648,Z 323.703,A -85,B 0,C 180,E1 -31640.336,E2 -31640.336} C_VEL
LIN {X 0,Y 51.39,Z 314.882,A -85,B 0,C 180,E1 -31641.528,E2 -31641.528} C_VEL
LIN {X 0,Y 54.141,Z 309.773,A -85,B 0,C 180,E1 -31642.808,E2 -31642.808} C_VEL
LIN {X 0,Y 57.661,Z 301.113,A -85,B 0,C 180,E1 -31646.288,E2 -31646.288} C_VEL
LIN {X 0,Y 60.654,Z 292.127,A -85,B 0,C 180,E1 -31649.286,E2 -31649.286} C_VEL
LIN {X 0,Y 62.416,Z 286.501,A -85,B 0,C 180,E1 -31649.935,E2 -31649.935} C_VEL
LIN {X 0,Y 65.912,Z 272.769,A -85,B 0,C 180,E1 -31650.128,E2 -31650.128} C_VEL
LIN {X 0,Y 67.725,Z 261.384,A -85,B 0,C 180,E1 -31650.347,E2 -31650.347} C_VEL
LIN {X 0,Y 67.425,Z 258.474,A -85,B 0,C 180,E1 -31654.948,E2 -31654.948} C_VEL
LIN {X 0,Y 67.408,Z 256.354,A -85,B 0,C 180,E1 -31661.774,E2 -31661.774} C_VEL
LIN {X 0,Y 67.487,Z 256.429,A -85,B 0,C 180,E1 -31664.462,E2 -31664.462} C_VEL
LIN {X 0,Y 67.563,Z 259.054,A -85,B 0,C 180,E1 -31668.849,E2 -31668.849} C_VEL
LIN {X 0,Y 67.787,Z 261.875,A -85,B 0,C 180,E1 -31672.283,E2 -31672.283} C_VEL
LIN {X 0,Y 65.262,Z 276.74,A -85,B 0,C 180,E1 -31672.473,E2 -31672.473} C_VEL
LIN {X 0,Y 62.015,Z 288.788,A -85,B 0,C 180,E1 -31672.586,E2 -31672.586} C_VEL
LIN {X 0,Y 57.511,Z 300.687,A -85,B 0,C 180,E1 -31672.608,E2 -31672.608} C_VEL
LIN {X 0,Y 50.895,Z 313.654,A -85,B 0,C 180,E1 -31672.598,E2 -31672.598} C_VEL
LIN {X 0,Y 43.404,Z 325.135,A -85,B 0,C 180,E1 -31672.638,E2 -31672.638} C_VEL
LIN {X 0,Y 35.428,Z 334.911,A -85,B 0,C 180,E1 -31672.688,E2 -31672.688} C_VEL
LIN {X 0,Y 26.576,Z 343.788,A -85,B 0,C 180,E1 -31672.6,E2 -31672.6} C_VEL
LIN {X 0,Y 17.702,Z 351.183,A -85,B 0,C 180,E1 -31672.995,E2 -31672.995} C_VEL
LIN {X 0,Y 7.076,Z 358.396,A -85,B 0,C 180,E1 -31673.325,E2 -31673.325} C_VEL
LIN {X 0,Y 5.477,Z 359.222,A -85,B 0,C 180,E1 -31655.315,E2 -31655.315} C_VEL
LIN {X 0,Y 16.443,Z 351.847,A -85,B 0,C 180,E1 -31648.743,E2 -31648.743} C_VEL
LIN {X 0,Y 27,Z 342.978,A -85,B 0,C 180,E1 -31648.632,E2 -31648.632} C_VEL
LIN {X 0,Y 35.91,Z 333.805,A -85,B 0,C 180,E1 -31648.898,E2 -31648.898} C_VEL
LIN {X 0,Y 43.992,Z 323.625,A -85,B 0,C 180,E1 -31649.17,E2 -31649.17} C_VEL
LIN {X 0,Y 51.715,Z 311.424,A -85,B 0,C 180,E1 -31649.44,E2 -31649.44} C_VEL
LIN {X 0,Y 57.507,Z 299.785,A -85,B 0,C 180,E1 -31649.669,E2 -31649.669} C_VEL
LIN {X 0,Y 62.204,Z 287.206,A -85,B 0,C 180,E1 -31649.898,E2 -31649.898} C_VEL
LIN {X 0,Y 62.416,Z 286.501,A -85,B 0,C 180,E1 -31649.935,E2 -31649.935} C_VEL
LIN {X 0,Y 63.445,Z 282.716,A -85,B 0,C 180,E1 -31650.538,E2 -31650.538} C_VEL
LIN {X 0,Y 64.545,Z 276.71,A -85,B 0,C 180,E1 -31653.112,E2 -31653.112} C_VEL
LIN {X 0,Y 65.488,Z 270.638,A -85,B 0,C 180,E1 -31655.635,E2 -31655.635} C_VEL
LIN {X 0,Y 66.071,Z 266.737,A -85,B 0,C 180,E1 -31656.226,E2 -31656.226} C_VEL
LIN {X 0,Y 66.262,Z 265.382,A -85,B 0,C 180,E1 -31656.355,E2 -31656.355} C_VEL
LIN {X 0,Y 66.292,Z 263.975,A -85,B 0,C 180,E1 -31660.267,E2 -31660.267} C_VEL
LIN {X 0,Y 66.389,Z 263.438,A -85,B 0,C 180,E1 -31663.284,E2 -31663.284} C_VEL
LIN {X 0,Y 66.298,Z 265.408,A -85,B 0,C 180,E1 -31666.303,E2 -31666.303} C_VEL
LIN {X 0,Y 63.731,Z 279.135,A -85,B 0,C 180,E1 -31666.226,E2 -31666.226} C_VEL
LIN {X 0,Y 60.308,Z 290.802,A -85,B 0,C 180,E1 -31665.945,E2 -31665.945} C_VEL
LIN {X 0,Y 55.25,Z 303.31,A -85,B 0,C 180,E1 -31665.369,E2 -31665.369} C_VEL
LIN {X 0,Y 49.247,Z 314.71,A -85,B 0,C 180,E1 -31664.426,E2 -31664.426} C_VEL
LIN {X 0,Y 42.233,Z 325.319,A -85,B 0,C 180,E1 -31663.109,E2 -31663.109} C_VEL
LIN {X 0,Y 37,Z 331.968,A -85,B 0,C 180,E1 -31661.757,E2 -31661.757} C_VEL
LIN {X 0,Y 37.45,Z 331.381,A -85,B 0,C 180,E1 -31659.773,E2 -31659.773} C_VEL
LIN {X 0,Y 45.448,Z 320.603,A -85,B 0,C 180,E1 -31658.1,E2 -31658.1} C_VEL
LIN {X 0,Y 52.427,Z 308.79,A -85,B 0,C 180,E1 -31657.162,E2 -31657.162} C_VEL
LIN {X 0,Y 58.436,Z 295.598,A -85,B 0,C 180,E1 -31656.562,E2 -31656.562} C_VEL
LIN {X 0,Y 62.811,Z 282.307,A -85,B 0,C 180,E1 -31656.398,E2 -31656.398} C_VEL
LIN {X 0,Y 65.671,Z 269.173,A -85,B 0,C 180,E1 -31656.244,E2 -31656.244} C_VEL
LIN {X 0,Y 66.071,Z 266.737,A -85,B 0,C 180,E1 -31656.226,E2 -31656.226} C_VEL
LIN {X 0,Y 70.05,Z 267.031,A -85,B 0,C 180,E1 -31656.237,E2 -31656.237} C_VEL
LIN {X 0,Y 70.05,Z 600,A -85,B 0,C 180,E1 -31656.237,E2 -31656.237} C_VEL
LIN {X 0,Y 70.05,Z 600,A -85,B 0,C 180,E1 -31656.237,E2 -31656.237}

QRS_NEXT_CUT()

QRS_NEXT()
QRS_HOME()

END
